C01820=1089.401,52.222,440.400,175.154,18.357,152.860
C01821=1089.407,52.472,440.384,175.156,18.358,152.860
C01822=1089.412,52.722,440.367,175.158,18.360,152.860
C01823=1089.418,52.971,440.351,175.160,18.362,152.860
C01824=1089.423,53.220,440.335,175.161,18.363,152.860
C01825=1089.429,53.469,440.319,175.163,18.365,152.860
C01826=1089.435,53.719,440.303,175.165,18.367,152.860
C01827=1089.441,53.969,440.287,175.167,18.368,152.860
C01828=1089.447,54.218,440.271,175.169,18.370,152.860
C01829=1089.453,54.467,440.255,175.171,18.372,152.860
C01830=1089.458,54.717,440.239,175.173,18.373,152.860
C01831=1089.464,54.966,440.223,175.175,18.375,152.860
C01832=1089.469,55.216,440.206,175.177,18.376,152.860
C01833=1089.475,55.465,440.190,175.178,18.378,152.860
C01834=1089.481,55.714,440.174,175.180,18.380,152.860
C01835=1089.486,55.964,440.158,175.182,18.381,152.860
C01836=1089.492,56.214,440.142,175.184,18.383,152.860
C01837=1089.498,56.463,440.126,175.186,18.385,152.860
C01838=1089.504,56.712,440.110,175.188,18.386,152.860
C01839=1089.510,56.961,440.094,175.189,18.388,152.860
C01840=1089.515,57.211,440.077,175.192,18.389,152.860
C01841=1089.521,57.460,440.061,175.193,18.391,152.860
C01842=1089.526,57.710,440.045,175.196,18.392,152.860
C01843=1089.532,57.959,440.029,175.197,18.394,152.860
C01844=1089.538,58.209,440.013,175.199,18.396,152.860
C01845=1089.544,58.458,439.996,175.201,18.397,152.860
C01846=1089.549,58.708,439.979,175.203,18.399,152.860
C01847=1089.555,58.957,439.963,175.205,18.400,152.859
C01848=1089.561,59.206,439.947,175.206,18.402,152.859
C01849=1089.567,59.456,439.931,175.209,18.403,152.859
C01850=1089.573,59.705,439.914,175.210,18.405,152.859
C01851=1089.579,59.954,439.898,175.213,18.407,152.859
C01852=1089.584,60.204,439.881,175.214,18.408,152.859
C01853=1089.590,60.453,439.865,175.217,18.410,152.859
C01854=1089.596,60.702,439.849,175.218,18.411,152.859
C01855=1089.602,60.951,439.833,175.221,18.413,152.859
C01856=1089.608,61.201,439.817,175.222,18.414,152.859
C01857=1089.613,61.450,439.800,175.224,18.415,152.859
C01858=1089.619,61.700,439.784,175.226,18.418,152.859
C01859=1089.625,61.949,439.767,175.228,18.419,152.859
C01860=1089.631,62.198,439.751,175.230,18.421,152.859
C01861=1089.636,62.448,439.734,175.232,18.422,152.859
C01862=1089.642,62.697,439.718,175.234,18.424,152.859
C01863=1089.648,62.947,439.702,175.235,18.425,152.859
C01864=1089.654,63.224,439.683,175.238,18.427,152.859
C01865=1089.661,63.501,439.665,175.240,18.429,152.859
C01866=1089.667,63.778,439.647,175.242,18.431,152.859
C01867=1089.674,64.055,439.629,175.244,18.432,152.859
C01868=1089.680,64.304,439.612,175.246,18.434,152.859
C01869=1089.685,64.554,439.596,175.248,18.435,152.859
C01870=1089.691,64.803,439.579,175.250,18.437,152.859
C01871=1089.697,65.052,439.562,175.252,18.438,152.858
C01872=1089.702,65.302,439.545,175.254,18.440,152.858
C01873=1089.708,65.551,439.529,175.256,18.441,152.858
C01874=1089.714,65.801,439.512,175.258,18.443,152.858
C01875=1089.720,66.050,439.496,175.260,18.444,152.858
C01876=1089.725,66.300,439.479,175.262,18.446,152.858
C01877=1089.731,66.548,439.462,175.264,18.447,152.858
C01878=1089.737,66.798,439.446,175.266,18.450,152.858
C01879=1089.742,67.047,439.429,175.268,18.451,152.858
C01880=1089.748,67.297,439.413,175.270,18.453,152.858
C01881=1089.753,67.546,439.396,175.271,18.454,152.858
C01882=1089.760,67.795,439.379,175.274,18.456,152.858
C01883=1089.765,68.045,439.362,175.275,18.457,152.858
C01884=1089.771,68.294,439.346,175.278,18.459,152.858
C01885=1089.776,68.544,439.329,175.279,18.460,152.858
C01886=1089.782,68.792,439.312,175.282,18.462,152.858
C01887=1089.788,69.043,439.295,175.283,18.463,152.858
C01888=1089.794,69.292,439.279,175.286,18.465,152.858
C01889=1089.799,69.542,439.262,175.287,18.466,152.858
C01890=1089.806,69.791,439.245,175.290,18.468,152.858
C01891=1089.811,70.040,439.228,175.291,18.469,152.858
C01892=1089.817,70.290,439.212,175.294,18.471,152.857
C01893=1089.822,70.539,439.194,175.295,18.473,152.858
C01894=1089.828,70.788,439.178,175.297,18.474,152.857
C01895=1089.833,71.038,439.161,175.299,18.476,152.857
C01896=1089.839,71.287,439.144,175.301,18.477,152.857
C01897=1089.845,71.536,439.127,175.303,18.478,152.857
C01898=1089.850,71.786,439.110,175.305,18.480,152.857
C01899=1089.856,72.034,439.093,175.307,18.482,152.857
C01900=1089.862,72.284,439.077,175.309,18.484,152.857
C01901=1089.867,72.534,439.060,175.311,18.485,152.857
C01902=1089.874,72.783,439.042,175.313,18.486,152.857
C01903=1089.879,73.033,439.026,175.315,18.488,152.857
C01904=1089.884,73.282,439.008,175.317,18.489,152.857
C01905=1089.890,73.531,438.992,175.319,18.491,152.857
C01906=1089.895,73.781,438.975,175.321,18.493,152.857
C01907=1089.902,74.030,438.958,175.323,18.494,152.857
C01908=1089.907,74.279,438.941,175.325,18.496,152.857
C01909=1089.912,74.528,438.923,175.327,18.497,152.857
C01910=1089.918,74.778,438.907,175.329,18.499,152.857
C01911=1089.924,75.027,438.890,175.331,18.500,152.857
C01912=1089.930,75.277,438.872,175.333,18.501,152.856
C01913=1089.936,75.526,438.855,175.335,18.503,152.856
C01914=1089.941,75.775,438.839,175.337,18.505,152.856
C01915=1089.947,76.024,438.821,175.339,18.506,152.856
C01916=1089.953,76.274,438.805,175.341,18.508,152.856
C01917=1089.958,76.523,438.787,175.343,18.509,152.856
C01918=1089.964,76.773,438.770,175.345,18.510,152.856
C01919=1089.970,77.022,438.752,175.347,18.512,152.856
C01920=1089.976,77.272,438.736,175.349,18.514,152.856
C01921=1089.981,77.521,438.719,175.352,18.515,152.856
C01922=1089.986,77.770,438.702,175.353,18.517,152.856
C01923=1089.992,78.019,438.685,175.355,18.518,152.856
C01924=1089.999,78.269,438.667,175.357,18.519,152.856
C01925=1090.004,78.518,438.650,175.360,18.521,152.855
C01926=1090.009,78.767,438.632,175.361,18.522,152.856
C01927=1090.015,79.017,438.616,175.364,18.524,152.855
C01928=1090.021,79.294,438.596,175.366,18.526,152.855
C01929=1090.028,79.571,438.577,175.367,18.527,152.855
C01930=1090.034,79.848,438.558,175.370,18.529,152.855
C01931=1090.040,80.124,438.539,175.372,18.531,152.855
C01932=1090.046,80.374,438.521,175.374,18.532,152.855
C01933=1090.051,80.623,438.504,175.376,18.533,152.855
C01934=1090.057,80.872,438.487,175.379,18.536,152.855
C01935=1090.062,81.121,438.469,175.380,18.537,152.855
C01936=1090.068,81.371,438.452,175.383,18.538,152.855
C01937=1090.073,81.620,438.435,175.384,18.539,152.855
C01938=1090.079,81.870,438.417,175.387,18.541,152.855
C01939=1090.084,82.119,438.400,175.388,18.542,152.855
C01940=1090.091,82.368,438.383,175.391,18.544,152.854
C01941=1090.096,82.617,438.366,175.392,18.546,152.855
C01942=1090.102,82.867,438.348,175.395,18.547,152.854
C01943=1090.108,83.117,438.331,175.396,18.548,152.854
C01944=1090.113,83.366,438.313,175.399,18.550,152.854
C01945=1090.119,83.615,438.296,175.401,18.552,152.854
C01946=1090.124,83.864,438.278,175.403,18.553,152.854
C01947=1090.130,84.114,438.261,175.405,18.554,152.854
C01948=1090.135,84.363,438.243,175.407,18.556,152.854
C01949=1090.141,84.612,438.226,175.410,18.557,152.854
C01950=1090.147,84.861,438.208,175.411,18.559,152.854
C01951=1090.153,85.111,438.190,175.413,18.560,152.854
C01952=1090.158,85.361,438.173,175.415,18.561,152.854
C01953=1090.163,85.610,438.156,175.418,18.563,152.853
C01954=1090.169,85.859,438.138,175.420,18.565,152.853
C01955=1090.175,86.108,438.120,175.421,18.566,152.853
C01956=1090.181,86.358,438.103,175.424,18.568,152.853
C01957=1090.186,86.607,438.085,175.426,18.569,152.853
C01958=1090.193,86.856,438.068,175.428,18.570,152.853
C01959=1090.198,87.106,438.051,175.430,18.571,152.853
C01960=1090.204,87.355,438.033,175.432,18.573,152.853
C01961=1090.210,87.604,438.016,175.434,18.574,152.853
C01962=1090.215,87.853,437.998,175.436,18.576,152.853
C01963=1090.221,88.102,437.980,175.439,18.578,152.853
C01964=1090.227,88.352,437.962,175.440,18.579,152.852
C01965=1090.232,88.601,437.945,175.443,18.580,152.852
C01966=1090.238,88.850,437.927,175.445,18.581,152.852
C01967=1090.244,89.100,437.909,175.447,18.583,152.852
C01968=1090.250,89.349,437.892,175.449,18.584,152.852
C01969=1090.255,89.598,437.874,175.451,18.586,152.852
C01970=1090.261,89.848,437.856,175.454,18.588,152.852
C01971=1090.266,90.097,437.838,175.455,18.589,152.852
C01972=1090.272,90.346,437.821,175.458,18.590,152.852
C01973=1090.278,90.596,437.803,175.459,18.591,152.852
C01974=1090.283,90.845,437.785,175.462,18.593,152.851
C01975=1090.289,91.095,437.767,175.464,18.594,152.851
C01976=1090.295,91.344,437.750,175.466,18.596,152.851
C01977=1090.300,91.593,437.732,175.469,18.597,152.851
C01978=1090.306,91.843,437.714,175.470,18.598,152.851
C01979=1090.311,92.092,437.696,175.473,18.600,152.851
C01980=1090.317,92.341,437.678,175.474,18.601,152.851
C01981=1090.323,92.591,437.660,175.477,18.603,152.851
C01982=1090.328,92.840,437.643,175.478,18.604,152.851
C01983=1090.334,93.088,437.625,175.481,18.606,152.851
C01984=1090.340,93.338,437.606,175.483,18.607,152.850
C01985=1090.345,93.587,437.588,175.485,18.608,152.850
C01986=1090.351,93.836,437.571,175.487,18.610,152.850
C01987=1090.357,94.086,437.553,175.489,18.611,152.850
C01988=1090.362,94.335,437.535,175.492,18.612,152.850
C01989=1090.368,94.585,437.517,175.494,18.614,152.850
C01990=1090.373,94.834,437.499,175.496,18.615,152.850
C01991=1090.379,95.083,437.481,175.498,18.617,152.850
C01992=1090.385,95.361,437.461,175.501,18.618,152.850
C01993=1090.391,95.637,437.440,175.503,18.620,152.849
C01994=1090.398,95.914,437.421,175.505,18.621,152.849
C01995=1090.404,96.190,437.401,175.507,18.623,152.849
C01996=1090.410,96.440,437.383,175.510,18.624,152.849
C01997=1090.415,96.690,437.365,175.512,18.625,152.849
C01998=1090.421,96.939,437.347,175.514,18.627,152.849
C01999=1090.427,97.188,437.328,175.517,18.628,152.849
C02000=1090.432,97.437,437.311,175.518,18.629,152.849
C02001=1090.438,97.687,437.292,175.521,18.631,152.848
C02002=1090.443,97.936,437.275,175.522,18.632,152.848
C02003=1090.450,98.185,437.256,175.525,18.634,152.848
C02004=1090.455,98.434,437.238,175.527,18.635,152.848
C02005=1090.461,98.684,437.220,175.529,18.636,152.848
C02006=1090.467,98.933,437.202,175.532,18.638,152.848
C02007=1090.472,99.183,437.183,175.533,18.639,152.848
C02008=1090.477,99.432,437.166,175.536,18.640,152.848
C02009=1090.484,99.681,437.147,175.538,18.642,152.848
C02010=1090.489,99.930,437.129,175.540,18.643,152.847
C02011=1090.495,100.180,437.111,175.542,18.645,152.847
C02012=1090.501,100.428,437.093,175.544,18.646,152.847
C02013=1090.507,100.678,437.075,175.547,18.647,152.847
C02014=1090.511,100.927,437.057,175.549,18.648,152.847
C02015=1090.518,101.176,437.038,175.551,18.649,152.847
C02016=1090.523,101.426,437.020,175.554,18.651,152.847
C02017=1090.529,101.675,437.001,175.556,18.653,152.847
C02018=1090.534,101.924,436.983,175.558,18.654,152.846
C02019=1090.540,102.174,436.965,175.560,18.655,152.846
C02020=1090.545,102.423,436.946,175.562,18.656,152.846
C02021=1090.551,102.672,436.928,175.564,18.658,152.846
C02022=1090.556,102.921,436.909,175.567,18.660,152.846
C02023=1090.562,103.171,436.891,175.569,18.661,152.846
C02024=1090.568,103.420,436.872,175.571,18.662,152.846
C02025=1090.574,103.669,436.855,175.574,18.664,152.846
C02026=1090.579,103.918,436.836,175.575,18.665,152.846
C02027=1090.585,104.168,436.818,175.578,18.666,152.845
C02028=1090.590,104.417,436.799,175.580,18.667,152.845
C02029=1090.596,104.666,436.781,175.582,18.669,152.845
C02030=1090.601,104.915,436.762,175.585,18.670,152.845
C02031=1090.607,105.165,436.744,175.586,18.671,152.845
C02032=1090.612,105.414,436.725,175.589,18.673,152.845
C02033=1090.618,105.663,436.707,175.591,18.674,152.845
C02034=1090.624,105.912,436.688,175.593,18.675,152.844
C02035=1090.630,106.161,436.670,175.596,18.676,152.844
C02036=1090.635,106.411,436.651,175.597,18.678,152.844
C02037=1090.640,106.660,436.632,175.600,18.679,152.844
C02038=1090.647,106.910,436.614,175.602,18.681,152.844
C02039=1090.652,107.158,436.596,175.604,18.682,152.844
C02040=1090.658,107.408,436.577,175.607,18.683,152.843
C02041=1090.663,107.657,436.559,175.609,18.684,152.843
C02042=1090.669,107.906,436.540,175.611,18.686,152.843
C02043=1090.675,108.156,436.522,175.614,18.687,152.843
C02044=1090.680,108.405,436.503,175.616,18.688,152.843
C02045=1090.686,108.654,436.484,175.618,18.689,152.843
C02046=1090.692,108.903,436.465,175.621,18.691,152.843
C02047=1090.697,109.152,436.447,175.622,18.692,152.843
C02048=1090.703,109.402,436.428,175.625,18.693,152.842
C02049=1090.708,109.651,436.409,175.627,18.695,152.842
C02050=1090.714,109.900,436.391,175.629,18.696,152.842
C02051=1090.720,110.150,436.372,175.632,18.697,152.842
C02052=1090.725,110.398,436.353,175.634,18.698,152.842
C02053=1090.731,110.648,436.334,175.636,18.699,152.842
C02054=1090.737,110.898,436.316,175.639,18.701,152.841
C02055=1090.743,111.146,436.298,175.641,18.702,152.841
C02056=1090.749,111.424,436.276,175.644,18.704,152.841
C02057=1090.755,111.700,436.256,175.645,18.705,152.841
C02058=1090.761,111.977,436.235,175.648,18.706,152.841
C02059=1090.768,112.255,436.214,175.651,18.707,152.841
C02060=1090.773,112.503,436.195,175.653,18.709,152.840
C02061=1090.779,112.753,436.176,175.656,18.711,152.840
C02062=1090.785,113.002,436.157,175.658,18.711,152.840
C02063=1090.790,113.251,436.138,175.660,18.713,152.840
C02064=1090.796,113.501,436.120,175.663,18.714,152.840
C02065=1090.801,113.750,436.101,175.665,18.715,152.840
C02066=1090.807,113.999,436.082,175.667,18.716,152.839
C02067=1090.813,114.248,436.063,175.670,18.718,152.839
C02068=1090.819,114.498,436.044,175.672,18.719,152.839
C02069=1090.824,114.746,436.025,175.674,18.720,152.839
C02070=1090.829,114.996,436.006,175.677,18.722,152.839
C02071=1090.835,115.245,435.986,175.678,18.723,152.839
C02072=1090.840,115.494,435.968,175.681,18.724,152.839
C02073=1090.846,115.744,435.949,175.683,18.725,152.838
C02074=1090.851,115.993,435.930,175.685,18.727,152.838
C02075=1090.856,116.242,435.911,175.688,18.728,152.838
C02076=1090.862,116.491,435.892,175.690,18.729,152.838
C02077=1090.868,116.741,435.873,175.692,18.730,152.838
C02078=1090.874,116.989,435.854,175.695,18.731,152.838
C02079=1090.879,117.239,435.835,175.697,18.733,152.837
C02080=1090.885,117.488,435.816,175.699,18.734,152.837
C02081=1090.890,117.737,435.797,175.701,18.736,152.837
C02082=1090.896,117.986,435.778,175.704,18.737,152.837
C02083=1090.901,118.236,435.758,175.706,18.738,152.837
C02084=1090.907,118.485,435.739,175.709,18.739,152.837
C02085=1090.912,118.734,435.720,175.711,18.740,152.836
C02086=1090.918,118.983,435.701,175.714,18.742,152.836
C02087=1090.924,119.233,435.682,175.716,18.743,152.836
C02088=1090.929,119.481,435.662,175.718,18.744,152.836
C02089=1090.935,119.730,435.643,175.721,18.746,152.836
C02090=1090.940,119.980,435.624,175.723,18.746,152.836
C02091=1090.946,120.229,435.604,175.725,18.748,152.835
C02092=1090.951,120.478,435.585,175.728,18.749,152.835
C02093=1090.957,120.727,435.566,175.729,18.750,152.835
C02094=1090.962,120.977,435.547,175.732,18.751,152.835
C02095=1090.968,121.226,435.528,175.735,18.753,152.835
C02096=1090.974,121.476,435.509,175.736,18.754,152.835
C02097=1090.979,121.724,435.489,175.739,18.755,152.834
C02098=1090.985,121.973,435.470,175.742,18.756,152.834
C02099=1090.991,122.223,435.450,175.744,18.757,152.834
C02100=1090.996,122.472,435.431,175.746,18.759,152.834
C02101=1091.002,122.722,435.412,175.749,18.760,152.834
C02102=1091.007,122.970,435.392,175.751,18.761,152.833
C02103=1091.013,123.219,435.373,175.753,18.762,152.833
C02104=1091.019,123.469,435.354,175.756,18.763,152.833
C02105=1091.024,123.718,435.335,175.758,18.765,152.833
C02106=1091.029,123.968,435.315,175.760,18.766,152.833
C02107=1091.035,124.216,435.295,175.763,18.767,152.833
C02108=1091.040,124.465,435.276,175.765,18.768,152.832
C02109=1091.046,124.715,435.257,175.767,18.769,152.832
C02110=1091.052,124.963,435.237,175.770,18.770,152.832
C02111=1091.058,125.213,435.218,175.773,18.772,152.832
C02112=1091.064,125.462,435.198,175.775,18.773,152.831
C02113=1091.069,125.712,435.179,175.777,18.774,152.831
C02114=1091.075,125.961,435.159,175.780,18.775,152.831
C02115=1091.080,126.209,435.140,175.782,18.776,152.831
C02116=1091.086,126.459,435.121,175.784,18.777,152.831
C02117=1091.092,126.708,435.101,175.787,18.778,152.831
C02118=1091.097,126.957,435.081,175.789,18.780,152.830
C02119=1091.103,127.206,435.061,175.792,18.781,152.830
C02120=1091.110,127.483,435.040,175.795,18.782,152.830
C02121=1091.116,127.760,435.018,175.797,18.783,152.830
C02122=1091.122,128.037,434.996,175.800,18.784,152.829
C02123=1091.128,128.315,434.975,175.803,18.786,152.829
C02124=1091.134,128.563,434.955,175.805,18.787,152.829
C02125=1091.139,128.812,434.936,175.807,18.788,152.829
C02126=1091.145,129.061,434.916,175.810,18.789,152.829
C02127=1091.151,129.311,434.897,175.813,18.790,152.828
C02128=1091.157,129.559,434.877,175.815,18.791,152.828
C02129=1091.163,129.809,434.857,175.817,18.792,152.828
C02130=1091.168,130.058,434.837,175.820,18.794,152.828
C02131=1091.174,130.307,434.818,175.822,18.794,152.828
C02132=1091.179,130.556,434.798,175.825,18.795,152.827
C02133=1091.185,130.806,434.778,175.827,18.796,152.827
C02134=1091.191,131.055,434.758,175.830,18.798,152.827
C02135=1091.197,131.304,434.739,175.832,18.799,152.827
C02136=1091.202,131.553,434.719,175.834,18.800,152.826
C02137=1091.208,131.803,434.699,175.837,18.801,152.826
C02138=1091.214,132.051,434.679,175.840,18.802,152.826
C02139=1091.219,132.301,434.660,175.842,18.803,152.826
C02140=1091.225,132.550,434.640,175.844,18.804,152.826
C02141=1091.231,132.799,434.620,175.847,18.806,152.825
C02142=1091.236,133.048,434.600,175.850,18.807,152.825
C02143=1091.242,133.297,434.580,175.852,18.807,152.825
C02144=1091.247,133.547,434.561,175.854,18.809,152.825
C02145=1091.253,133.795,434.541,175.857,18.810,152.825
C02146=1091.259,134.045,434.520,175.859,18.811,152.824
C02147=1091.264,134.294,434.501,175.861,18.812,152.824
C02148=1091.270,134.543,434.480,175.864,18.813,152.824
C02149=1091.276,134.792,434.460,175.867,18.814,152.824
C02150=1091.281,135.041,434.441,175.869,18.815,152.823
C02151=1091.286,135.291,434.420,175.871,18.816,152.823
C02152=1091.292,135.539,434.401,175.874,18.818,152.823
C02153=1091.297,135.789,434.381,175.877,18.819,152.823
C02154=1091.303,136.038,434.361,175.879,18.819,152.823
C02155=1091.309,136.287,434.341,175.881,18.821,152.822
C02156=1091.315,136.536,434.320,175.884,18.822,152.822
C02157=1091.320,136.785,434.301,175.887,18.823,152.822
C02158=1091.326,137.034,434.280,175.889,18.824,152.822
C02159=1091.332,137.283,434.260,175.891,18.825,152.821
C02160=1091.337,137.532,434.240,175.894,18.826,152.821
C02161=1091.343,137.782,434.221,175.897,18.827,152.821
C02162=1091.348,138.031,434.200,175.899,18.829,152.821
C02163=1091.354,138.280,434.180,175.901,18.829,152.820
C02164=1091.360,138.529,434.160,175.904,18.830,152.820
C02165=1091.365,138.778,434.140,175.907,18.832,152.820
C02166=1091.371,139.027,434.120,175.909,18.833,152.820
C02167=1091.377,139.277,434.099,175.911,18.833,152.820
C02168=1091.382,139.526,434.079,175.914,18.835,152.819
C02169=1091.388,139.775,434.059,175.917,18.836,152.819
C02170=1091.393,140.024,434.038,175.919,18.837,152.819
C02171=1091.399,140.273,434.018,175.921,18.837,152.819
C02172=1091.404,140.522,433.998,175.924,18.839,152.818
C02173=1091.410,140.771,433.978,175.927,18.840,152.818
C02174=1091.415,141.020,433.958,175.929,18.841,152.818
C02175=1091.421,141.269,433.938,175.932,18.842,152.818
C02176=1091.427,141.518,433.918,175.934,18.843,152.817
C02177=1091.432,141.768,433.897,175.937,18.844,152.817
C02178=1091.438,142.016,433.877,175.939,18.845,152.817
C02179=1091.444,142.266,433.856,175.942,18.847,152.817
C02180=1091.449,142.515,433.836,175.944,18.847,152.817
C02181=1091.455,142.764,433.816,175.947,18.848,152.816
C02182=1091.460,143.013,433.795,175.950,18.849,152.816
C02183=1091.465,143.262,433.775,175.952,18.850,152.816
C02184=1091.472,143.539,433.752,175.955,18.852,152.815
C02185=1091.478,143.816,433.730,175.958,18.853,152.815
C02186=1091.485,144.093,433.707,175.961,18.854,152.815
C02187=1091.490,144.369,433.684,175.963,18.855,152.815
C02188=1091.497,144.619,433.664,175.966,18.856,152.814
C02189=1091.502,144.868,433.643,175.969,18.857,152.814
C02190=1091.507,145.117,433.622,175.972,18.858,152.814
C02191=1091.513,145.366,433.602,175.973,18.859,152.814
C02192=1091.519,145.615,433.582,175.976,18.860,152.813
C02193=1091.524,145.864,433.561,175.979,18.861,152.813
C02194=1091.530,146.114,433.540,175.982,18.862,152.813
C02195=1091.536,146.363,433.520,175.984,18.863,152.813
C02196=1091.541,146.611,433.499,175.986,18.864,152.812
C02197=1091.547,146.860,433.479,175.989,18.865,152.812
C02198=1091.553,147.109,433.459,175.992,18.866,152.812
C02199=1091.558,147.359,433.438,175.995,18.867,152.812
C02200=1091.564,147.608,433.417,175.997,18.868,152.811
C02201=1091.569,147.857,433.397,175.999,18.869,152.811
C02202=1091.575,148.105,433.376,176.002,18.870,152.811
C02203=1091.581,148.355,433.355,176.005,18.871,152.811
C02204=1091.586,148.604,433.335,176.008,18.872,152.810
C02205=1091.592,148.853,433.314,176.010,18.873,152.810
C02206=1091.597,149.103,433.293,176.013,18.874,152.810
C02207=1091.603,149.351,433.273,176.015,18.875,152.810
C02208=1091.609,149.601,433.252,176.018,18.876,152.809
C02209=1091.614,149.850,433.231,176.021,18.877,152.809
C02210=1091.620,150.098,433.210,176.023,18.878,152.809
C02211=1091.625,150.347,433.189,176.026,18.879,152.808
C02212=1091.631,150.597,433.169,176.028,18.880,152.808
C02213=1091.636,150.846,433.148,176.031,18.881,152.808
C02214=1091.642,151.095,433.127,176.033,18.882,152.808
C02215=1091.648,151.344,433.107,176.036,18.883,152.807
C02216=1091.654,151.593,433.086,176.039,18.884,152.807
C02217=1091.659,151.842,433.065,176.042,18.885,152.807
C02218=1091.664,152.091,433.044,176.044,18.886,152.807
C02219=1091.670,152.340,433.023,176.046,18.887,152.806
C02220=1091.676,152.589,433.002,176.049,18.888,152.806
C02221=1091.681,152.839,432.981,176.052,18.889,152.806
C02222=1091.687,153.087,432.960,176.055,18.890,152.806
C02223=1091.692,153.336,432.939,176.057,18.891,152.805
C02224=1091.698,153.586,432.919,176.060,18.891,152.805
C02225=1091.703,153.834,432.897,176.062,18.893,152.805
C02226=1091.709,154.084,432.877,176.065,18.894,152.804
C02227=1091.715,154.333,432.855,176.068,18.895,152.804
C02228=1091.720,154.582,432.835,176.071,18.896,152.804
C02229=1091.726,154.830,432.813,176.073,18.897,152.804
C02230=1091.731,155.080,432.792,176.075,18.898,152.803
C02231=1091.737,155.329,432.771,176.078,18.898,152.803
C02232=1091.742,155.578,432.750,176.081,18.899,152.803
C02233=1091.748,155.827,432.729,176.084,18.900,152.803
C02234=1091.754,156.076,432.708,176.087,18.902,152.802
C02235=1091.759,156.325,432.687,176.089,18.903,152.802
C02236=1091.765,156.575,432.666,176.092,18.904,152.802
C02237=1091.771,156.823,432.645,176.094,18.904,152.802
C02238=1091.776,157.072,432.624,176.097,18.905,152.801
C02239=1091.782,157.321,432.603,176.100,18.906,152.801
C02240=1091.787,157.571,432.582,176.102,18.907,152.801
C02241=1091.793,157.819,432.561,176.105,18.908,152.800
C02242=1091.799,158.068,432.539,176.108,18.909,152.800
C02243=1091.804,158.317,432.519,176.111,18.910,152.800
C02244=1091.809,158.566,432.497,176.113,18.911,152.799
C02245=1091.815,158.816,432.476,176.116,18.912,152.799
C02246=1091.821,159.065,432.455,176.118,18.913,152.799
C02247=1091.827,159.314,432.433,176.121,18.914,152.799
C02248=1091.833,159.590,432.409,176.124,18.915,152.798
C02249=1091.839,159.867,432.387,176.127,18.916,152.798
C02250=1091.845,160.143,432.363,176.131,18.917,152.798
C02251=1091.852,160.420,432.339,176.134,18.918,152.797
C02252=1091.857,160.669,432.318,176.136,18.919,152.797
C02253=1091.863,160.918,432.296,176.138,18.920,152.797
C02254=1091.869,161.167,432.275,176.141,18.920,152.796
C02255=1091.874,161.416,432.253,176.144,18.921,152.796
C02256=1091.879,161.666,432.232,176.147,18.922,152.796
C02257=1091.885,161.914,432.211,176.149,18.924,152.796
C02258=1091.890,162.164,432.189,176.152,18.925,152.795
C02259=1091.896,162.412,432.168,176.155,18.925,152.795
C02260=1091.901,162.661,432.147,176.158,18.926,152.795
C02261=1091.907,162.911,432.125,176.161,18.927,152.794
C02262=1091.912,163.159,432.104,176.163,18.928,152.794
C02263=1091.918,163.408,432.082,176.165,18.929,152.794
C02264=1091.923,163.657,432.060,176.168,18.930,152.794
C02265=1091.928,163.906,432.039,176.171,18.931,152.793
C02266=1091.934,164.156,432.017,176.174,18.932,152.793
C02267=1091.939,164.404,431.996,176.177,18.933,152.793
C02268=1091.944,164.653,431.974,176.179,18.934,152.792
C02269=1091.950,164.902,431.952,176.182,18.935,152.792
C02270=1091.956,165.151,431.931,176.185,18.936,152.792
C02271=1091.961,165.400,431.909,176.187,18.937,152.792
C02272=1091.967,165.649,431.888,176.190,18.938,152.791
C02273=1091.972,165.898,431.865,176.193,18.939,152.791
C02274=1091.978,166.148,431.845,176.196,18.939,152.791
C02275=1091.982,166.396,431.823,176.198,18.940,152.790
C02276=1091.989,166.646,431.801,176.201,18.942,152.790
C02277=1091.993,166.894,431.780,176.204,18.943,152.790
C02278=1092.000,167.144,431.758,176.207,18.943,152.789
C02279=1092.005,167.392,431.737,176.210,18.944,152.789
C02280=1092.011,167.642,431.714,176.212,18.946,152.789
C02281=1092.016,167.890,431.693,176.215,18.946,152.789
C02282=1092.022,168.140,431.671,176.217,18.947,152.788
C02283=1092.027,168.388,431.650,176.220,18.948,152.788
C02284=1092.033,168.638,431.627,176.223,18.949,152.788
C02285=1092.038,168.886,431.606,176.226,18.950,152.787
C02286=1092.044,169.136,431.584,176.229,18.951,152.787
C02287=1092.049,169.384,431.563,176.232,18.951,152.787
C02288=1092.055,169.633,431.540,176.234,18.952,152.786
C02289=1092.060,169.882,431.518,176.237,18.954,152.786
C02290=1092.066,170.131,431.496,176.240,18.954,152.786
C02291=1092.071,170.380,431.475,176.243,18.955,152.786
C02292=1092.077,170.629,431.453,176.246,18.956,152.785
C02293=1092.083,170.878,431.431,176.249,18.957,152.785
C02294=1092.088,171.127,431.409,176.251,18.958,152.785
C02295=1092.093,171.377,431.387,176.253,18.958,152.784
C02296=1092.099,171.625,431.365,176.256,18.959,152.784
C02297=1092.105,171.874,431.343,176.259,18.961,152.784
C02298=1092.110,172.123,431.321,176.262,18.961,152.783
C02299=1092.116,172.372,431.299,176.265,18.962,152.783
C02300=1092.122,172.621,431.278,176.268,18.963,152.783
C02301=1092.127,172.869,431.255,176.271,18.964,152.782
C02302=1092.133,173.119,431.233,176.274,18.965,152.782
C02303=1092.138,173.368,431.211,176.276,18.966,152.782
C02304=1092.143,173.617,431.189,176.279,18.967,152.782
C02305=1092.150,173.866,431.167,176.282,18.968,152.781
C02306=1092.155,174.114,431.145,176.285,18.969,152.781
C02307=1092.161,174.364,431.123,176.288,18.969,152.780
C02308=1092.166,174.613,431.101,176.291,18.970,152.780
C02309=1092.171,174.861,431.079,176.294,18.971,152.780
C02310=1092.177,175.111,431.057,176.296,18.972,152.780
C02311=1092.183,175.360,431.035,176.298,18.972,152.779
C02312=1092.189,175.636,431.011,176.302,18.973,152.779
C02313=1092.195,175.911,430.986,176.305,18.974,152.778
C02314=1092.202,176.188,430.961,176.308,18.975,152.778
C02315=1092.208,176.464,430.936,176.312,18.976,152.778
C02316=1092.214,176.714,430.915,176.315,18.977,152.777
C02317=1092.219,176.963,430.892,176.317,18.978,152.777
C02318=1092.224,177.211,430.870,176.320,18.979,152.777
C02319=1092.231,177.460,430.848,176.323,18.979,152.776
C02320=1092.236,177.710,430.825,176.326,18.980,152.776
C02321=1092.241,177.958,430.803,176.328,18.981,152.776
C02322=1092.247,178.207,430.781,176.331,18.982,152.775
C02323=1092.253,178.456,430.759,176.334,18.983,152.775
C02324=1092.259,178.705,430.736,176.337,18.983,152.775
C02325=1092.264,178.954,430.715,176.340,18.984,152.774
C02326=1092.270,179.203,430.692,176.343,18.985,152.774
C02327=1092.275,179.452,430.669,176.346,18.986,152.774
C02328=1092.282,179.701,430.647,176.349,18.987,152.773
C02329=1092.287,179.950,430.625,176.352,18.988,152.773
C02330=1092.292,180.199,430.602,176.355,18.988,152.773
C02331=1092.298,180.448,430.581,176.357,18.989,152.772
C02332=1092.304,180.697,430.558,176.360,18.990,152.772
C02333=1092.310,180.946,430.535,176.363,18.991,152.771
C02334=1092.316,181.194,430.514,176.366,18.992,152.771
C02335=1092.321,181.443,430.491,176.369,18.992,152.771
C02336=1092.327,181.692,430.468,176.372,18.993,152.770
C02337=1092.332,181.941,430.445,176.375,18.994,152.770
C02338=1092.339,182.190,430.423,176.378,18.995,152.770
C02339=1092.344,182.439,430.401,176.381,18.995,152.769
C02340=1092.349,182.688,430.378,176.384,18.996,152.769
C02341=1092.355,182.937,430.355,176.387,18.997,152.769
C02342=1092.361,183.186,430.334,176.390,18.998,152.768
C02343=1092.367,183.435,430.311,176.393,18.998,152.768
C02344=1092.373,183.684,430.288,176.395,19.000,152.768
C02345=1092.378,183.933,430.266,176.398,19.000,152.767
C02346=1092.384,184.181,430.244,176.401,19.001,152.767
C02347=1092.390,184.430,430.221,176.404,19.001,152.766
C02348=1092.396,184.679,430.198,176.407,19.003,152.766
C02349=1092.401,184.928,430.175,176.410,19.003,152.766
C02350=1092.407,185.177,430.152,176.413,19.004,152.765
C02351=1092.412,185.426,430.130,176.416,19.004,152.765
C02352=1092.418,185.675,430.107,176.419,19.006,152.765
C02353=1092.423,185.924,430.085,176.422,19.006,152.764
C02354=1092.429,186.173,430.062,176.425,19.007,152.764
C02355=1092.434,186.422,430.039,176.428,19.008,152.764
C02356=1092.440,186.670,430.016,176.430,19.009,152.763
C02357=1092.445,186.919,429.993,176.433,19.010,152.763
C02358=1092.451,187.168,429.971,176.436,19.010,152.763
C02359=1092.456,187.417,429.948,176.439,19.012,152.762
C02360=1092.461,187.666,429.925,176.442,19.012,152.762
C02361=1092.467,187.915,429.902,176.445,19.013,152.762
C02362=1092.473,188.164,429.879,176.448,19.014,152.761
C02363=1092.478,188.412,429.856,176.451,19.015,152.761
C02364=1092.484,188.661,429.833,176.454,19.016,152.761
C02365=1092.489,188.910,429.810,176.457,19.016,152.760
C02366=1092.495,189.160,429.788,176.460,19.017,152.760
C02367=1092.500,189.409,429.764,176.462,19.018,152.760
C02368=1092.506,189.658,429.742,176.465,19.019,152.759
C02369=1092.511,189.906,429.719,176.468,19.020,152.759
C02370=1092.517,190.155,429.696,176.471,19.021,152.759
C02371=1092.522,190.404,429.673,176.474,19.021,152.758
C02372=1092.528,190.653,429.650,176.477,19.022,152.758
C02373=1092.533,190.902,429.627,176.480,19.023,152.757
C02374=1092.539,191.151,429.604,176.483,19.024,152.757
C02375=1092.544,191.400,429.581,176.486,19.024,152.757
C02376=1092.550,191.675,429.555,176.490,19.025,152.756
C02377=1092.557,191.951,429.530,176.492,19.027,152.756
C02378=1092.563,192.227,429.504,176.496,19.028,152.756
C02379=1092.569,192.503,429.478,176.499,19.028,152.755
C02380=1092.575,192.751,429.455,176.502,19.029,152.755
C02381=1092.580,193.000,429.432,176.505,19.030,152.754
C02382=1092.585,193.249,429.409,176.508,19.031,152.754
C02383=1092.591,193.498,429.386,176.511,19.031,152.754
C02384=1092.597,193.747,429.363,176.514,19.032,152.753
C02385=1092.603,193.996,429.340,176.517,19.033,152.753
C02386=1092.608,194.245,429.316,176.520,19.033,152.753
C02387=1092.614,194.493,429.293,176.523,19.034,152.752
C02388=1092.619,194.742,429.270,176.526,19.035,152.752
C02389=1092.625,194.991,429.247,176.530,19.036,152.751
C02390=1092.630,195.240,429.223,176.533,19.037,152.751
C02391=1092.636,195.489,429.200,176.535,19.038,152.751
C02392=1092.642,195.737,429.177,176.538,19.039,152.750
C02393=1092.648,195.986,429.154,176.541,19.039,152.750
C02394=1092.653,196.236,429.130,176.544,19.040,152.750
C02395=1092.658,196.484,429.107,176.547,19.041,152.749
C02396=1092.664,196.733,429.084,176.550,19.041,152.749
C02397=1092.669,196.982,429.060,176.553,19.042,152.749
C02398=1092.675,197.231,429.037,176.556,19.043,152.748
C02399=1092.681,197.480,429.014,176.559,19.044,152.748
C02400=1092.687,197.729,428.990,176.562,19.044,152.747
C02401=1092.692,197.978,428.967,176.565,19.045,152.747
C02402=1092.698,198.227,428.944,176.569,19.046,152.747
C02403=1092.704,198.475,428.920,176.572,19.047,152.746
C02404=1092.709,198.724,428.896,176.575,19.048,152.746
C02405=1092.715,198.973,428.873,176.578,19.049,152.746
C02406=1092.721,199.222,428.850,176.581,19.049,152.745
C02407=1092.726,199.471,428.826,176.584,19.050,152.745
C02408=1092.732,199.719,428.803,176.587,19.051,152.744
C02409=1092.738,199.968,428.780,176.590,19.051,152.744
C02410=1092.743,200.217,428.756,176.593,19.052,152.744
C02411=1092.749,200.466,428.732,176.596,19.053,152.743
C02412=1092.754,200.715,428.709,176.599,19.053,152.743
C02413=1092.760,200.964,428.685,176.602,19.054,152.742
C02414=1092.766,201.212,428.662,176.605,19.055,152.742
C02415=1092.771,201.461,428.638,176.608,19.056,152.742
C02416=1092.777,201.710,428.615,176.611,19.057,152.741
C02417=1092.784,201.959,428.591,176.614,19.058,152.741
C02418=1092.789,202.208,428.567,176.617,19.058,152.741
C02419=1092.795,202.456,428.544,176.620,19.059,152.740
C02420=1092.800,202.706,428.520,176.623,19.059,152.740
C02421=1092.806,202.954,428.496,176.626,19.060,152.739
C02422=1092.811,203.203,428.473,176.629,19.061,152.739
C02423=1092.817,203.451,428.449,176.633,19.062,152.739
C02424=1092.823,203.701,428.425,176.636,19.063,152.738
C02425=1092.828,203.950,428.401,176.639,19.063,152.738
C02426=1092.834,204.198,428.377,176.642,19.064,152.737
C02427=1092.839,204.447,428.354,176.645,19.065,152.737
C02428=1092.845,204.696,428.330,176.648,19.066,152.737
C02429=1092.850,204.944,428.306,176.651,19.066,152.736
C02430=1092.855,205.193,428.282,176.654,19.067,152.736
C02431=1092.862,205.442,428.258,176.657,19.068,152.735
C02432=1092.867,205.691,428.234,176.660,19.069,152.735
C02433=1092.873,205.940,428.211,176.663,19.070,152.735
C02434=1092.878,206.188,428.187,176.666,19.071,152.734
C02435=1092.883,206.437,428.163,176.669,19.071,152.734
C02436=1092.890,206.686,428.139,176.672,19.072,152.734
C02437=1092.895,206.935,428.115,176.675,19.073,152.733
C02438=1092.900,207.184,428.091,176.679,19.074,152.733
C02439=1092.906,207.432,428.067,176.682,19.075,152.732
C02440=1092.929,208.451,427.969,176.741,19.102,152.728
C02441=1092.937,208.827,427.932,176.746,19.104,152.727
C02442=1092.946,209.204,427.896,176.750,19.107,152.727
C02443=1092.955,209.581,427.858,176.755,19.109,152.727
C02444=1092.963,209.957,427.822,176.759,19.112,152.727
C02445=1092.969,210.206,427.797,176.762,19.113,152.727
C02446=1092.974,210.455,427.773,176.765,19.115,152.726
C02447=1092.980,210.703,427.748,176.768,19.117,152.726
C02448=1092.986,210.952,427.724,176.771,19.119,152.726
C02449=1092.991,211.201,427.700,176.774,19.120,152.726
C02450=1092.997,211.450,427.675,176.777,19.121,152.726
C02451=1093.002,211.699,427.651,176.780,19.124,152.726
C02452=1093.008,211.947,427.626,176.782,19.125,152.726
C02453=1093.014,212.196,427.601,176.786,19.127,152.725
C02454=1093.019,212.445,427.577,176.789,19.128,152.725
C02455=1093.024,212.693,427.553,176.792,19.130,152.725
C02456=1093.030,212.943,427.528,176.795,19.132,152.725
C02457=1093.036,213.191,427.503,176.798,19.134,152.725
C02458=1093.042,213.440,427.478,176.801,19.135,152.724
C02459=1093.047,213.688,427.454,176.803,19.137,152.724
C02460=1093.053,213.938,427.430,176.807,19.139,152.724
C02461=1093.058,214.186,427.405,176.809,19.140,152.724
C02462=1093.064,214.434,427.380,176.813,19.142,152.724
C02463=1093.070,214.684,427.356,176.815,19.144,152.724
C02464=1093.075,214.932,427.331,176.819,19.145,152.723
C02465=1093.081,215.181,427.306,176.821,19.147,152.723
C02466=1093.086,215.429,427.282,176.824,19.149,152.723
C02467=1093.091,215.678,427.257,176.827,19.150,152.723
C02468=1093.097,215.927,427.232,176.831,19.152,152.723
C02469=1093.103,216.176,427.207,176.833,19.154,152.723
C02470=1093.108,216.425,427.183,176.837,19.156,152.722
C02471=1093.114,216.673,427.158,176.839,19.157,152.722
C02472=1093.120,216.922,427.133,176.842,19.159,152.722
C02473=1093.126,217.170,427.108,176.845,19.161,152.722
C02474=1093.131,217.420,427.083,176.848,19.162,152.722
C02475=1093.136,217.668,427.058,176.851,19.164,152.722
C02476=1093.142,217.917,427.033,176.854,19.165,152.722
C02477=1093.148,218.166,427.009,176.857,19.168,152.721
C02478=1093.154,218.414,426.984,176.860,19.169,152.721
C02479=1093.159,218.663,426.960,176.863,19.171,152.721
C02480=1093.164,218.912,426.934,176.866,19.173,152.721
C02481=1093.170,219.160,426.909,176.869,19.175,152.721
C02482=1093.176,219.409,426.884,176.872,19.176,152.721
C02483=1093.181,219.658,426.860,176.875,19.178,152.720
C02484=1093.187,219.906,426.834,176.878,19.179,152.720
C02485=1093.193,220.155,426.808,176.881,19.181,152.720
C02486=1093.198,220.404,426.784,176.884,19.183,152.720
C02487=1093.204,220.653,426.759,176.887,19.185,152.720
C02488=1093.210,220.901,426.735,176.890,19.186,152.720
C02489=1093.215,221.150,426.709,176.893,19.188,152.720
C02490=1093.221,221.398,426.684,176.896,19.189,152.719
C02491=1093.227,221.647,426.659,176.899,19.192,152.719
C02492=1093.233,221.896,426.634,176.902,19.193,152.719
C02493=1093.241,222.277,426.595,176.907,19.196,152.719
C02494=1093.250,222.657,426.556,176.911,19.198,152.718
C02495=1093.258,223.038,426.518,176.916,19.201,152.718
C02496=1093.267,223.418,426.480,176.921,19.204,152.718
C02497=1093.272,223.667,426.454,176.923,19.205,152.718
C02498=1093.278,223.915,426.429,176.927,19.207,152.718
C02499=1093.283,224.164,426.403,176.929,19.209,152.718
C02500=1093.289,224.412,426.378,176.933,19.211,152.717
C02501=1093.294,224.662,426.353,176.935,19.212,152.717
C02502=1093.300,224.910,426.328,176.939,19.214,152.717
C02503=1093.305,225.159,426.302,176.941,19.216,152.717
C02504=1093.311,225.407,426.277,176.945,19.218,152.717
C02505=1093.317,225.656,426.252,176.947,19.219,152.717
C02506=1093.322,225.904,426.226,176.950,19.221,152.717
C02507=1093.328,226.154,426.201,176.953,19.223,152.716
C02508=1093.334,226.403,426.176,176.957,19.225,152.716
C02509=1093.339,226.651,426.151,176.960,19.227,152.716
C02510=1093.345,226.900,426.125,176.963,19.228,152.716
C02511=1093.351,227.148,426.099,176.966,19.230,152.716
C02512=1093.356,227.397,426.074,176.968,19.232,152.716
C02513=1093.362,227.645,426.048,176.972,19.233,152.715
C02514=1093.368,227.894,426.022,176.975,19.235,152.715
C02515=1093.373,228.142,425.997,176.978,19.237,152.715
C02516=1093.379,228.391,425.972,176.981,19.238,152.715
C02517=1093.385,228.640,425.946,176.984,19.240,152.715
C02518=1093.390,228.889,425.920,176.986,19.242,152.715
C02519=1093.395,229.137,425.895,176.990,19.244,152.715
C02520=1093.401,229.386,425.869,176.993,19.245,152.714
C02521=1093.407,229.635,425.843,176.996,19.247,152.714
C02522=1093.413,229.883,425.818,176.999,19.249,152.714
C02523=1093.418,230.132,425.793,177.002,19.251,152.714
C02524=1093.424,230.380,425.767,177.005,19.253,152.714
C02525=1093.430,230.629,425.741,177.008,19.254,152.714
C02526=1093.435,230.878,425.715,177.011,19.256,152.713
C02527=1093.441,231.126,425.690,177.014,19.258,152.713
C02528=1093.446,231.375,425.664,177.017,19.260,152.713
C02529=1093.452,231.624,425.638,177.020,19.261,152.713
C02530=1093.458,231.872,425.612,177.023,19.263,152.713
C02531=1093.463,232.121,425.587,177.027,19.265,152.713
C02532=1093.468,232.370,425.561,177.029,19.267,152.713
C02533=1093.474,232.619,425.535,177.033,19.269,152.712
C02534=1093.480,232.867,425.510,177.035,19.270,152.712
C02535=1093.486,233.116,425.483,177.038,19.272,152.712
C02536=1093.491,233.364,425.457,177.042,19.275,152.712
C02537=1093.497,233.612,425.432,177.045,19.276,152.712
C02538=1093.502,233.861,425.406,177.048,19.278,152.712
C02539=1093.508,234.110,425.380,177.050,19.280,152.712
C02540=1093.514,234.359,425.354,177.054,19.282,152.712
C02541=1093.519,234.607,425.328,177.056,19.283,152.711
C02542=1093.525,234.855,425.302,177.060,19.285,152.711
C02543=1093.531,235.104,425.276,177.063,19.287,152.711
C02544=1093.536,235.353,425.250,177.066,19.289,152.711
C02545=1093.544,235.725,425.211,177.071,19.291,152.711
C02546=1093.553,236.097,425.172,177.075,19.294,152.711
C02547=1093.561,236.469,425.134,177.079,19.297,152.710
C02548=1093.569,236.840,425.094,177.084,19.300,152.710
C02549=1093.575,237.089,425.068,177.087,19.301,152.710
C02550=1093.580,237.338,425.042,177.090,19.303,152.710
C02551=1093.586,237.587,425.015,177.094,19.305,152.710
C02552=1093.592,237.835,424.990,177.096,19.307,152.710
C02553=1093.597,238.083,424.963,177.100,19.309,152.709
C02554=1093.603,238.332,424.938,177.102,19.310,152.709
C02555=1093.609,238.580,424.911,177.106,19.313,152.709
C02556=1093.614,238.829,424.885,177.109,19.315,152.709
C02557=1093.620,239.078,424.858,177.112,19.316,152.709
C02558=1093.625,239.327,424.832,177.115,19.318,152.709
C02559=1093.631,239.575,424.806,177.117,19.320,152.709
C02560=1093.637,239.823,424.779,177.121,19.322,152.709
C02561=1093.642,240.072,424.753,177.124,19.323,152.708
C02562=1093.648,240.321,424.727,177.127,19.325,152.708
C02563=1093.654,240.570,424.701,177.130,19.327,152.708
C02564=1093.659,240.818,424.674,177.134,19.329,152.708
C02565=1093.665,241.066,424.647,177.136,19.331,152.708
C02566=1093.671,241.315,424.621,177.140,19.333,152.708
C02567=1093.676,241.564,424.595,177.142,19.334,152.708
C02568=1093.681,241.812,424.569,177.145,19.336,152.707
C02569=1093.688,242.061,424.542,177.149,19.339,152.707
C02570=1093.693,242.310,424.515,177.152,19.340,152.707
C02571=1093.699,242.558,424.489,177.155,19.342,152.707
C02572=1093.705,242.807,424.463,177.158,19.344,152.707
C02573=1093.711,243.055,424.436,177.161,19.346,152.707
C02574=1093.716,243.304,424.410,177.164,19.347,152.707
C02575=1093.722,243.552,424.383,177.167,19.349,152.706
C02576=1093.727,243.800,424.357,177.170,19.351,152.706
C02577=1093.732,244.049,424.330,177.173,19.353,152.706
C02578=1093.738,244.297,424.303,177.176,19.355,152.706
C02579=1093.744,244.546,424.277,177.179,19.357,152.706
C02580=1093.749,244.795,424.251,177.183,19.359,152.706
C02581=1093.755,245.043,424.224,177.185,19.361,152.706
C02582=1093.760,245.292,424.197,177.189,19.362,152.706
C02583=1093.766,245.541,424.170,177.192,19.365,152.705
C02584=1093.772,245.789,424.143,177.195,19.366,152.705
C02585=1093.778,246.037,424.117,177.198,19.368,152.705
C02586=1093.783,246.286,424.090,177.201,19.370,152.705
C02587=1093.789,246.534,424.063,177.204,19.372,152.705
C02588=1093.794,246.783,424.036,177.207,19.374,152.705
C02589=1093.800,247.032,424.010,177.211,19.376,152.705
C02590=1093.806,247.280,423.984,177.213,19.377,152.705
C02591=1093.811,247.529,423.956,177.217,19.380,152.704
C02592=1093.816,247.777,423.930,177.220,19.382,152.704
C02593=1093.822,248.026,423.903,177.222,19.383,152.704
C02594=1093.827,248.274,423.876,177.226,19.386,152.704
C02595=1093.833,248.523,423.849,177.229,19.388,152.704
C02596=1093.838,248.771,423.822,177.232,19.389,152.704
C02597=1093.847,249.136,423.783,177.237,19.392,152.704
C02598=1093.855,249.501,423.743,177.241,19.395,152.704
C02599=1093.863,249.866,423.703,177.246,19.398,152.704
C02600=1093.871,250.231,423.663,177.250,19.401,152.703
C02601=1093.877,250.479,423.636,177.253,19.403,152.703
C02602=1093.882,250.728,423.609,177.256,19.405,152.703
C02603=1093.888,250.976,423.582,177.259,19.407,152.703
C02604=1093.893,251.225,423.555,177.262,19.409,152.703
C02605=1093.899,251.474,423.528,177.266,19.411,152.703
C02606=1093.904,251.722,423.500,177.268,19.413,152.703
C02607=1093.910,251.970,423.474,177.272,19.415,152.703
C02608=1093.915,252.219,423.446,177.275,19.417,152.703
C02609=1093.921,252.467,423.420,177.278,19.418,152.702
C02610=1093.926,252.716,423.392,177.281,19.421,152.702
C02611=1093.932,252.964,423.365,177.284,19.423,152.702
C02612=1093.938,253.213,423.338,177.288,19.425,152.702
C02613=1093.943,253.462,423.311,177.290,19.426,152.702
C02614=1093.949,253.710,423.283,177.293,19.429,152.702
C02615=1093.955,253.958,423.256,177.297,19.431,152.702
C02616=1093.960,254.207,423.229,177.299,19.432,152.702
C02617=1093.966,254.455,423.201,177.303,19.434,152.702
C02618=1093.971,254.704,423.174,177.306,19.437,152.701
C02619=1093.977,254.952,423.147,177.309,19.439,152.701
C02620=1093.982,255.200,423.119,177.312,19.440,152.701
C02621=1093.988,255.449,423.093,177.315,19.443,152.701
C02622=1093.994,255.698,423.065,177.319,19.445,152.701
C02623=1094.000,255.946,423.038,177.321,19.446,152.701
C02624=1094.005,256.194,423.010,177.324,19.448,152.701
C02625=1094.011,256.442,422.983,177.328,19.451,152.701
C02626=1094.017,256.691,422.956,177.331,19.453,152.701
C02627=1094.022,256.939,422.928,177.334,19.454,152.701
C02628=1094.028,257.188,422.901,177.337,19.456,152.700
C02629=1094.034,257.437,422.873,177.340,19.459,152.700
C02630=1094.040,257.685,422.846,177.344,19.461,152.700
C02631=1094.045,257.933,422.818,177.346,19.462,152.700
C02632=1094.050,258.182,422.791,177.350,19.464,152.700
C02633=1094.057,258.430,422.763,177.353,19.466,152.700
C02634=1094.062,258.679,422.736,177.355,19.468,152.700
C02635=1094.068,258.927,422.708,177.359,19.470,152.700
C02636=1094.074,259.175,422.680,177.362,19.472,152.699
C02637=1094.079,259.424,422.653,177.365,19.474,152.699
C02638=1094.085,259.672,422.625,177.368,19.476,152.699
C02639=1094.090,259.921,422.598,177.371,19.478,152.699
C02640=1094.096,260.169,422.570,177.375,19.480,152.699
C02641=1094.102,260.418,422.542,177.378,19.482,152.699
C02642=1094.107,260.666,422.515,177.380,19.484,152.699
C02643=1094.113,260.914,422.487,177.384,19.486,152.699
C02644=1094.119,261.163,422.459,177.387,19.488,152.699
C02645=1094.125,261.411,422.431,177.391,19.490,152.699
C02646=1094.130,261.659,422.404,177.393,19.492,152.699
C02647=1094.137,261.908,422.376,177.396,19.494,152.698
C02648=1094.142,262.156,422.348,177.400,19.496,152.698
C02649=1094.151,262.518,422.308,177.404,19.499,152.698
C02650=1094.159,262.881,422.267,177.409,19.502,152.698
C02651=1094.167,263.242,422.227,177.413,19.504,152.698
C02652=1094.176,263.605,422.186,177.418,19.508,152.698
C02653=1094.181,263.853,422.158,177.422,19.510,152.698
C02654=1094.188,264.101,422.131,177.424,19.511,152.697
C02655=1094.193,264.350,422.103,177.427,19.514,152.697
C02656=1094.199,264.598,422.074,177.431,19.516,152.697
C02657=1094.204,264.846,422.046,177.434,19.518,152.697
C02658=1094.210,265.094,422.018,177.437,19.520,152.697
C02659=1094.216,265.343,421.990,177.440,19.522,152.697
C02660=1094.221,265.592,421.963,177.443,19.524,152.697
C02661=1094.227,265.841,421.935,177.446,19.526,152.697
C02662=1094.232,266.089,421.907,177.450,19.529,152.697
C02663=1094.238,266.337,421.878,177.453,19.531,152.697
C02664=1094.243,266.585,421.850,177.456,19.532,152.697
C02665=1094.248,266.833,421.822,177.459,19.534,152.697
C02666=1094.254,267.082,421.794,177.462,19.537,152.697
C02667=1094.260,267.330,421.766,177.465,19.539,152.696
C02668=1094.266,267.578,421.737,177.469,19.541,152.696
C02669=1094.271,267.826,421.709,177.471,19.543,152.696
C02670=1094.277,268.075,421.681,177.475,19.545,152.696
C02671=1094.283,268.323,421.653,177.478,19.547,152.696
C02672=1094.289,268.572,421.624,177.481,19.549,152.696
C02673=1094.294,268.820,421.596,177.485,19.552,152.696
C02674=1094.300,269.069,421.568,177.487,19.554,152.696
C02675=1094.305,269.317,421.540,177.490,19.556,152.696
C02676=1094.311,269.566,421.512,177.494,19.558,152.696
C02677=1094.317,269.813,421.483,177.497,19.560,152.696
C02678=1094.323,270.062,421.455,177.500,19.562,152.696
C02679=1094.328,270.310,421.427,177.503,19.564,152.695
C02680=1094.334,270.559,421.399,177.506,19.566,152.696
C02681=1094.340,270.806,421.370,177.509,19.569,152.695
C02682=1094.345,271.055,421.341,177.512,19.571,152.695
C02683=1094.351,271.304,421.313,177.516,19.573,152.695
C02684=1094.356,271.552,421.285,177.519,19.575,152.695
C02685=1094.362,271.800,421.256,177.521,19.577,152.695
C02686=1094.368,272.048,421.228,177.525,19.579,152.695
C02687=1094.374,272.297,421.199,177.528,19.581,152.695
C02688=1094.379,272.544,421.171,177.531,19.584,152.695
C02689=1094.385,272.793,421.142,177.535,19.586,152.695
C02690=1094.390,273.041,421.114,177.538,19.588,152.695
C02691=1094.396,273.289,421.085,177.540,19.590,152.695
C02692=1094.402,273.538,421.056,177.544,19.592,152.695
C02693=1094.407,273.786,421.029,177.547,19.594,152.695
C02694=1094.413,274.035,420.999,177.550,19.597,152.695
C02695=1094.418,274.283,420.971,177.554,19.599,152.695
C02696=1094.425,274.531,420.942,177.557,19.601,152.694
C02697=1094.430,274.780,420.913,177.559,19.603,152.695
C02698=1094.435,275.027,420.884,177.562,19.605,152.694
C02699=1094.441,275.276,420.856,177.566,19.608,152.694
C02700=1094.447,275.524,420.827,177.569,19.610,152.694
C02701=1094.455,275.890,420.785,177.574,19.613,152.694
C02702=1094.463,276.254,420.743,177.578,19.616,152.694
C02703=1094.472,276.619,420.700,177.583,19.620,152.694
C02704=1094.480,276.984,420.658,177.588,19.623,152.694
C02705=1094.486,277.232,420.629,177.591,19.626,152.694
C02706=1094.491,277.480,420.601,177.593,19.627,152.694
C02707=1094.497,277.729,420.571,177.597,19.629,152.694
C02708=1094.503,277.977,420.542,177.600,19.632,152.694
C02709=1094.508,278.225,420.514,177.603,19.634,152.694
C02710=1094.514,278.473,420.484,177.607,19.636,152.694
C02711=1094.520,278.721,420.455,177.610,19.639,152.694
C02712=1094.525,278.970,420.426,177.613,19.641,152.694
C02713=1094.531,279.218,420.398,177.616,19.643,152.694
C02714=1094.537,279.466,420.369,177.619,19.645,152.694
C02715=1094.542,279.715,420.340,177.622,19.647,152.694
C02716=1094.548,279.962,420.311,177.625,19.649,152.693
C02717=1094.553,280.211,420.282,177.628,19.652,152.693
C02718=1094.560,280.459,420.252,177.632,19.654,152.693
C02719=1094.565,280.708,420.224,177.635,19.657,152.693
C02720=1094.570,280.955,420.195,177.638,19.659,152.693
C02721=1094.576,281.204,420.165,177.642,19.661,152.693
C02722=1094.582,281.452,420.136,177.645,19.664,152.693
C02723=1094.588,281.700,420.107,177.648,19.666,152.693
C02724=1094.593,281.948,420.078,177.650,19.668,152.693
C02725=1094.599,282.197,420.049,177.654,19.670,152.693
C02726=1094.604,282.445,420.019,177.657,19.673,152.693
C02727=1094.610,282.693,419.991,177.660,19.675,152.693
C02728=1094.615,282.941,419.961,177.663,19.677,152.693
C02729=1094.621,283.190,419.931,177.666,19.680,152.693
C02730=1094.627,283.438,419.902,177.670,19.682,152.693
C02731=1094.632,283.686,419.873,177.673,19.684,152.693
C02732=1094.638,283.934,419.844,177.676,19.687,152.693
C02733=1094.644,284.182,419.814,177.679,19.689,152.693
C02734=1094.649,284.431,419.785,177.682,19.692,152.693
C02735=1094.655,284.679,419.756,177.685,19.693,152.693
C02736=1094.660,284.926,419.726,177.688,19.696,152.693
C02737=1094.666,285.175,419.697,177.691,19.698,152.693
C02738=1094.672,285.423,419.668,177.695,19.701,152.693
C02739=1094.678,285.671,419.638,177.698,19.703,152.693
C02740=1094.683,285.920,419.609,177.701,19.705,152.693
C02741=1094.688,286.168,419.579,177.704,19.708,152.693
C02742=1094.695,286.415,419.549,177.707,19.710,152.693
C02743=1094.700,286.664,419.520,177.711,19.712,152.693
C02744=1094.706,286.912,419.490,177.714,19.715,152.693
C02745=1094.712,287.160,419.461,177.717,19.717,152.693
C02746=1094.717,287.409,419.432,177.720,19.720,152.693
C02747=1094.723,287.657,419.402,177.724,19.722,152.693
C02748=1094.728,287.906,419.372,177.727,19.724,152.693
C02749=1094.734,288.152,419.343,177.730,19.727,152.693
C02750=1094.740,288.401,419.313,177.732,19.729,152.693
C02751=1094.745,288.649,419.284,177.735,19.731,152.693
C02752=1094.751,288.898,419.254,177.739,19.733,152.693
C02753=1094.760,289.272,419.209,177.744,19.737,152.693
C02754=1094.769,289.646,419.165,177.748,19.741,152.693
C02755=1094.777,290.020,419.119,177.753,19.744,152.693
C02756=1094.785,290.394,419.074,177.758,19.748,152.693
C02757=1094.792,290.643,419.045,177.761,19.751,152.693
C02758=1094.798,290.890,419.015,177.764,19.753,152.693
C02759=1094.803,291.139,418.985,177.768,19.755,152.693
C02760=1094.809,291.387,418.956,177.771,19.758,152.693
C02761=1094.814,291.635,418.925,177.774,19.760,152.693
C02762=1094.819,291.883,418.896,177.777,19.763,152.693
C02763=1094.825,292.131,418.866,177.780,19.765,152.693
C02764=1094.831,292.379,418.836,177.784,19.768,152.693
C02765=1094.836,292.627,418.806,177.787,19.770,152.693
C02766=1094.842,292.875,418.776,177.790,19.773,152.693
C02767=1094.848,293.123,418.746,177.793,19.775,152.693
C02768=1094.853,293.372,418.716,177.796,19.778,152.693
C02769=1094.859,293.620,418.686,177.799,19.780,152.693
C02770=1094.865,293.868,418.656,177.802,19.783,152.693
C02771=1094.870,294.116,418.626,177.806,19.785,152.693
C02772=1094.876,294.364,418.596,177.809,19.787,152.693
C02773=1094.882,294.612,418.566,177.812,19.790,152.693
C02774=1094.888,294.860,418.535,177.815,19.793,152.693
C02775=1094.893,295.108,418.506,177.818,19.795,152.693
C02776=1094.899,295.356,418.475,177.822,19.797,152.693
C02777=1094.905,295.604,418.445,177.825,19.800,152.693
C02778=1094.910,295.852,418.415,177.828,19.803,152.693
C02779=1094.916,296.100,418.385,177.831,19.805,152.693
C02780=1094.922,296.348,418.355,177.834,19.807,152.693
C02781=1094.927,296.596,418.325,177.837,19.810,152.693
C02782=1094.933,296.844,418.295,177.840,19.813,152.693
C02783=1094.938,297.092,418.264,177.844,19.815,152.693
C02784=1094.944,297.342,418.234,177.847,19.818,152.693
C02785=1094.950,297.589,418.203,177.850,19.820,152.693
C02786=1094.956,297.837,418.173,177.853,19.823,152.694
C02787=1094.962,298.085,418.143,177.856,19.825,152.693
C02788=1094.968,298.333,418.112,177.859,19.828,152.694
C02789=1094.972,298.582,418.082,177.862,19.830,152.694
C02790=1094.978,298.829,418.052,177.866,19.833,152.694
C02791=1094.984,299.077,418.021,177.869,19.836,152.694
C02792=1094.989,299.325,417.990,177.872,19.838,152.694
C02793=1094.995,299.573,417.960,177.875,19.841,152.694
C02794=1095.001,299.821,417.930,177.878,19.844,152.694
C02795=1095.006,300.069,417.899,177.882,19.847,152.694
C02796=1095.011,300.318,417.869,177.885,19.849,152.694
C02797=1095.017,300.565,417.839,177.888,19.852,152.694
C02798=1095.022,300.814,417.808,177.891,19.855,152.694
C02799=1095.028,301.061,417.777,177.894,19.857,152.694
C02800=1095.033,301.310,417.747,177.897,19.860,152.694
C02801=1095.039,301.557,417.716,177.900,19.862,152.694
C02802=1095.045,301.806,417.685,177.903,19.865,152.694
C02803=1095.050,302.054,417.655,177.907,19.868,152.695
C02804=1095.056,302.302,417.624,177.910,19.870,152.695
C02805=1095.065,302.690,417.576,177.915,19.875,152.695
C02806=1095.074,303.078,417.528,177.920,19.879,152.695
C02807=1095.082,303.466,417.480,177.924,19.883,152.695
C02808=1095.091,303.854,417.432,177.930,19.887,152.695
C02809=1095.097,304.102,417.401,177.933,19.890,152.695
C02810=1095.103,304.350,417.370,177.936,19.893,152.695
C02811=1095.108,304.598,417.339,177.939,19.896,152.695
C02812=1095.113,304.846,417.308,177.942,19.898,152.695
C02813=1095.119,305.094,417.278,177.945,19.901,152.696
C02814=1095.125,305.342,417.246,177.948,19.903,152.696
C02815=1095.131,305.590,417.216,177.951,19.906,152.696
C02816=1095.136,305.838,417.185,177.954,19.909,152.696
C02817=1095.142,306.086,417.154,177.958,19.912,152.696
C02818=1095.147,306.333,417.123,177.961,19.915,152.696
C02819=1095.154,306.582,417.092,177.964,19.917,152.696
C02820=1095.159,306.830,417.061,177.967,19.920,152.696
C02821=1095.165,307.078,417.031,177.971,19.923,152.696
C02822=1095.170,307.325,416.999,177.974,19.925,152.696
C02823=1095.176,307.574,416.968,177.977,19.928,152.696
C02824=1095.182,307.821,416.937,177.980,19.931,152.696
C02825=1095.188,308.069,416.906,177.983,19.933,152.697
C02826=1095.193,308.318,416.875,177.987,19.937,152.697
C02827=1095.199,308.565,416.844,177.990,19.939,152.697
C02828=1095.205,308.813,416.813,177.993,19.942,152.697
C02829=1095.211,309.062,416.781,177.996,19.945,152.697
C02830=1095.216,309.310,416.751,177.999,19.947,152.697
C02831=1095.221,309.558,416.720,178.002,19.950,152.697
C02832=1095.228,309.806,416.688,178.005,19.953,152.697
C02833=1095.233,310.054,416.657,178.008,19.956,152.697
C02834=1095.239,310.301,416.626,178.012,19.959,152.697
C02835=1095.245,310.550,416.595,178.015,19.961,152.697
C02836=1095.250,310.797,416.563,178.018,19.964,152.698
C02837=1095.257,311.044,416.532,178.021,19.967,152.698
C02838=1095.262,311.293,416.501,178.024,19.970,152.698
C02839=1095.268,311.541,416.469,178.027,19.972,152.698
C02840=1095.274,311.789,416.438,178.030,19.975,152.698
C02841=1095.279,312.037,416.407,178.033,19.978,152.698
C02842=1095.285,312.285,416.376,178.037,19.981,152.698
C02843=1095.291,312.533,416.344,178.040,19.984,152.698
C02844=1095.297,312.780,416.313,178.043,19.987,152.698
C02845=1095.303,313.029,416.282,178.046,19.989,152.699
C02846=1095.308,313.276,416.250,178.050,19.992,152.699
C02847=1095.314,313.525,416.218,178.052,19.995,152.699
C02848=1095.319,313.773,416.187,178.056,19.997,152.699
C02849=1095.326,314.021,416.156,178.060,20.001,152.699
C02850=1095.332,314.268,416.124,178.062,20.004,152.699
C02851=1095.338,314.516,416.092,178.066,20.006,152.699
C02852=1095.343,314.764,416.062,178.068,20.009,152.699
C02853=1095.349,315.012,416.030,178.072,20.012,152.699
C02854=1095.355,315.260,415.998,178.075,20.014,152.700
C02855=1095.361,315.508,415.966,178.078,20.018,152.700
C02856=1095.366,315.756,415.935,178.081,20.021,152.700
C02857=1095.375,316.147,415.884,178.086,20.025,152.700
C02858=1095.384,316.538,415.835,178.091,20.030,152.700
C02859=1095.392,316.928,415.785,178.096,20.035,152.701
C02860=1095.401,317.319,415.734,178.101,20.039,152.701
C02861=1095.407,317.567,415.702,178.104,20.042,152.701
C02862=1095.412,317.815,415.671,178.107,20.046,152.701
C02863=1095.418,318.062,415.639,178.110,20.049,152.702
C02864=1095.423,318.311,415.608,178.113,20.052,152.702
C02865=1095.429,318.559,415.576,178.116,20.055,152.702
C02866=1095.435,318.807,415.544,178.119,20.058,152.702
C02867=1095.440,319.054,415.512,178.123,20.061,152.702
C02868=1095.446,319.303,415.480,178.126,20.064,152.702
C02869=1095.452,319.549,415.448,178.129,20.067,152.702
C02870=1095.457,319.798,415.415,178.132,20.070,152.703
C02871=1095.463,320.046,415.383,178.135,20.073,152.703
C02872=1095.468,320.294,415.352,178.138,20.077,152.703
C02873=1095.474,320.542,415.320,178.141,20.080,152.703
C02874=1095.480,320.789,415.288,178.144,20.082,152.703
C02875=1095.486,321.038,415.256,178.147,20.085,152.704
C02876=1095.491,321.285,415.224,178.151,20.089,152.704
C02877=1095.496,321.534,415.192,178.154,20.092,152.704
C02878=1095.502,321.781,415.160,178.157,20.095,152.704
C02879=1095.508,322.029,415.127,178.160,20.098,152.704
C02880=1095.514,322.277,415.095,178.163,20.101,152.704
C02881=1095.519,322.524,415.063,178.167,20.104,152.705
C02882=1095.525,322.773,415.031,178.169,20.107,152.705
C02883=1095.531,323.021,414.998,178.172,20.110,152.705
C02884=1095.536,323.268,414.966,178.175,20.113,152.705
C02885=1095.542,323.516,414.934,178.179,20.117,152.706
C02886=1095.548,323.764,414.903,178.182,20.120,152.706
C02887=1095.553,324.012,414.869,178.185,20.123,152.706
C02888=1095.559,324.260,414.837,178.188,20.126,152.706
C02889=1095.565,324.507,414.806,178.191,20.129,152.706
C02890=1095.571,324.755,414.773,178.194,20.132,152.707
C02891=1095.576,325.004,414.740,178.197,20.135,152.707
C02892=1095.582,325.252,414.708,178.201,20.139,152.707
C02893=1095.588,325.499,414.676,178.204,20.142,152.707
C02894=1095.594,325.747,414.644,178.207,20.145,152.707
C02895=1095.599,325.995,414.611,178.210,20.148,152.708
C02896=1095.605,326.242,414.579,178.213,20.152,152.708
C02897=1095.611,326.490,414.546,178.216,20.155,152.708
C02898=1095.617,326.738,414.514,178.219,20.158,152.708
C02899=1095.622,326.987,414.482,178.222,20.161,152.708
C02900=1095.628,327.234,414.449,178.226,20.164,152.709
C02901=1095.634,327.482,414.417,178.229,20.167,152.709
C02902=1095.640,327.730,414.384,178.232,20.170,152.709
C02903=1095.646,327.977,414.351,178.235,20.174,152.709
C02904=1095.652,328.225,414.319,178.238,20.177,152.710
C02905=1095.657,328.473,414.286,178.241,20.180,152.710
C02906=1095.663,328.721,414.254,178.244,20.183,152.710
C02907=1095.669,328.968,414.221,178.248,20.187,152.710
C02908=1095.675,329.216,414.188,178.251,20.190,152.710
C02909=1095.684,329.600,414.138,178.256,20.195,152.711
C02910=1095.693,329.984,414.087,178.260,20.200,152.711
C02911=1095.701,330.368,414.036,178.265,20.205,152.711
C02912=1095.711,330.751,413.986,178.270,20.210,152.712
C02913=1095.716,330.999,413.953,178.273,20.213,152.712
C02914=1095.722,331.247,413.920,178.276,20.216,152.712
C02915=1095.728,331.495,413.888,178.280,20.220,152.713
C02916=1095.734,331.743,413.855,178.282,20.223,152.713
C02917=1095.740,331.991,413.822,178.285,20.226,152.713
C02918=1095.746,332.239,413.789,178.289,20.230,152.713
C02919=1095.752,332.486,413.756,178.292,20.233,152.714
C02920=1095.757,332.734,413.724,178.295,20.237,152.714
C02921=1095.762,332.982,413.691,178.298,20.240,152.714
C02922=1095.769,333.229,413.658,178.301,20.244,152.715
C02923=1095.774,333.477,413.624,178.305,20.247,152.715
C02924=1095.780,333.725,413.591,178.307,20.251,152.715
C02925=1095.786,333.973,413.558,178.310,20.254,152.715
C02926=1095.792,334.221,413.525,178.314,20.258,152.716
C02927=1095.797,334.468,413.492,178.317,20.261,152.716
C02928=1095.803,334.716,413.459,178.319,20.264,152.716
C02929=1095.808,334.963,413.426,178.323,20.268,152.716
C02930=1095.814,335.211,413.393,178.326,20.271,152.717
C02931=1095.820,335.459,413.360,178.329,20.275,152.717
C02932=1095.826,335.707,413.327,178.332,20.278,152.717
C02933=1095.831,335.955,413.293,178.335,20.282,152.718
C02934=1095.837,336.203,413.260,178.338,20.285,152.718
C02935=1095.843,336.450,413.227,178.341,20.289,152.718
C02936=1095.849,336.698,413.194,178.345,20.292,152.718
C02937=1095.854,336.946,413.160,178.348,20.296,152.719
C02938=1095.860,337.194,413.127,178.350,20.299,152.719
C02939=1095.866,337.442,413.094,178.354,20.303,152.719
C02940=1095.872,337.689,413.061,178.357,20.306,152.720
C02941=1095.878,337.937,413.027,178.360,20.310,152.720
C02942=1095.883,338.185,412.994,178.363,20.313,152.720
C02943=1095.889,338.432,412.961,178.366,20.317,152.721
C02944=1095.895,338.680,412.928,178.369,20.321,152.721
C02945=1095.900,338.928,412.894,178.372,20.324,152.721
C02946=1095.906,339.175,412.860,178.376,20.328,152.722
C02947=1095.912,339.423,412.827,178.378,20.331,152.722
C02948=1095.917,339.671,412.794,178.382,20.335,152.722
C02949=1095.923,339.919,412.760,178.385,20.339,152.723
C02950=1095.929,340.166,412.726,178.388,20.343,152.723
C02951=1095.934,340.414,412.693,178.391,20.346,152.723
C02952=1095.940,340.662,412.659,178.393,20.350,152.724
C02953=1095.946,340.909,412.625,178.397,20.354,152.724
C02954=1095.951,341.157,412.592,178.400,20.357,152.724
C02955=1095.958,341.405,412.559,178.403,20.361,152.725
C02956=1095.964,341.652,412.525,178.406,20.364,152.725
C02957=1095.969,341.900,412.492,178.410,20.368,152.725
C02958=1095.975,342.147,412.458,178.412,20.371,152.726
C02959=1095.981,342.395,412.425,178.416,20.375,152.726
C02960=1095.986,342.643,412.390,178.419,20.379,152.726
C02961=1095.995,343.021,412.339,178.423,20.385,152.727
C02962=1096.003,343.399,412.288,178.428,20.391,152.728
C02963=1096.012,343.776,412.236,178.433,20.396,152.728
C02964=1096.021,344.154,412.185,178.438,20.402,152.729
C02965=1096.027,344.402,412.151,178.440,20.406,152.729
C02966=1096.033,344.649,412.117,178.443,20.409,152.729
C02967=1096.039,344.898,412.083,178.447,20.413,152.730
C02968=1096.045,345.145,412.049,178.450,20.418,152.730
C02969=1096.050,345.393,412.016,178.453,20.421,152.731
C02970=1096.055,345.640,411.981,178.456,20.425,152.731
C02971=1096.061,345.888,411.947,178.459,20.428,152.731
C02972=1096.067,346.135,411.914,178.462,20.433,152.732
C02973=1096.073,346.383,411.880,178.465,20.436,152.732
C02974=1096.078,346.630,411.846,178.468,20.440,152.733
C02975=1096.085,346.878,411.811,178.471,20.444,152.733
C02976=1096.090,347.126,411.777,178.474,20.448,152.733
C02977=1096.096,347.374,411.743,178.477,20.452,152.734
C02978=1096.101,347.621,411.709,178.480,20.456,152.734
C02979=1096.107,347.868,411.675,178.483,20.460,152.735
C02980=1096.112,348.116,411.641,178.486,20.464,152.735
C02981=1096.119,348.364,411.607,178.489,20.467,152.736
C02982=1096.124,348.612,411.573,178.492,20.472,152.736
C02983=1096.130,348.859,411.539,178.496,20.476,152.736
C02984=1096.135,349.106,411.504,178.498,20.480,152.737
C02985=1096.142,349.354,411.470,178.502,20.484,152.737
C02986=1096.148,349.602,411.436,178.504,20.488,152.738
C02987=1096.153,349.849,411.401,178.508,20.492,152.738
C02988=1096.159,350.097,411.367,178.510,20.496,152.739
C02989=1096.165,350.344,411.333,178.514,20.499,152.739
C02990=1096.170,350.592,411.298,178.516,20.503,152.740
C02991=1096.176,350.839,411.264,178.520,20.508,152.740
C02992=1096.182,351.087,411.230,178.523,20.512,152.740
C02993=1096.187,351.334,411.195,178.526,20.516,152.741
C02994=1096.194,351.582,411.161,178.529,20.520,152.741
C02995=1096.200,351.830,411.127,178.532,20.524,152.742
C02996=1096.205,352.077,411.092,178.535,20.528,152.742
C02997=1096.211,352.325,411.058,178.538,20.532,152.743
C02998=1096.216,352.573,411.023,178.541,20.536,152.743
C02999=1096.222,352.820,410.989,178.544,20.540,152.744
C03000=1096.228,353.067,410.955,178.547,20.544,152.744
C03001=1096.234,353.316,410.920,178.550,20.549,152.745
C03002=1096.240,353.562,410.885,178.554,20.553,152.745
C03003=1096.245,353.810,410.850,178.556,20.556,152.745
C03004=1096.251,354.058,410.816,178.560,20.561,152.746
C03005=1096.257,354.305,410.781,178.563,20.565,152.746
C03006=1096.262,354.553,410.747,178.565,20.569,152.747
C03007=1096.268,354.800,410.712,178.569,20.574,152.747
C03008=1096.274,355.048,410.677,178.571,20.577,152.748
C03009=1096.279,355.295,410.643,178.574,20.582,152.749
C03010=1096.285,355.543,410.607,178.578,20.586,152.749
C03011=1096.291,355.790,410.573,178.580,20.590,152.750
C03012=1096.296,356.038,410.538,178.584,20.595,152.750
C03013=1096.306,356.418,410.485,178.588,20.601,152.751
C03014=1096.315,356.798,410.432,178.593,20.608,152.752
C03015=1096.323,357.178,410.377,178.597,20.614,152.752
C03016=1096.332,357.558,410.324,178.602,20.621,152.753
C03017=1096.338,357.806,410.289,178.605,20.625,152.754
C03018=1096.344,358.053,410.255,178.608,20.630,152.754
C03019=1096.350,358.302,410.220,178.611,20.634,152.755
C03020=1096.355,358.549,410.184,178.614,20.638,152.755
C03021=1096.362,358.796,410.149,178.617,20.643,152.756
C03022=1096.367,359.044,410.114,178.620,20.647,152.756
C03023=1096.372,359.290,410.079,178.623,20.651,152.757
C03024=1096.379,359.538,410.045,178.626,20.656,152.758
C03025=1096.384,359.785,410.009,178.629,20.660,152.758
C03026=1096.390,360.034,409.974,178.632,20.664,152.759
C03027=1096.396,360.280,409.940,178.635,20.669,152.759
C03028=1096.402,360.528,409.904,178.638,20.673,152.760
C03029=1096.407,360.776,409.869,178.641,20.678,152.760
C03030=1096.413,361.023,409.833,178.644,20.682,152.761
C03031=1096.419,361.270,409.798,178.647,20.687,152.762
C03032=1096.425,361.518,409.764,178.650,20.691,152.762
C03033=1096.431,361.765,409.728,178.653,20.696,152.763
C03034=1096.436,362.012,409.693,178.656,20.700,152.763
C03035=1096.442,362.260,409.657,178.659,20.705,152.764
C03036=1096.447,362.508,409.623,178.662,20.710,152.764
C03037=1096.453,362.755,409.587,178.665,20.714,152.765
C03038=1096.460,363.002,409.552,178.668,20.719,152.766
C03039=1096.466,363.250,409.516,178.671,20.723,152.766
C03040=1096.472,363.497,409.481,178.674,20.728,152.767
C03041=1096.477,363.744,409.445,178.676,20.732,152.767
C03042=1096.483,363.992,409.409,178.680,20.737,152.768
C03043=1096.488,364.239,409.375,178.683,20.741,152.769
C03044=1096.494,364.487,409.339,178.686,20.746,152.769
C03045=1096.500,364.734,409.304,178.688,20.750,152.770
C03046=1096.506,364.981,409.269,178.691,20.755,152.771
C03047=1096.512,365.228,409.233,178.695,20.760,152.771
C03048=1096.518,365.476,409.198,178.698,20.765,152.772
C03049=1096.524,365.724,409.162,178.701,20.770,152.772
C03050=1096.529,365.971,409.126,178.703,20.774,152.773
C03051=1096.535,366.218,409.091,178.706,20.779,152.774
C03052=1096.541,366.465,409.055,178.709,20.784,152.774
C03053=1096.546,366.713,409.019,178.712,20.789,152.775
C03054=1096.551,366.960,408.984,178.716,20.793,152.776
C03055=1096.558,367.207,408.947,178.718,20.798,152.776
C03056=1096.563,367.454,408.912,178.721,20.803,152.777
C03057=1096.569,367.702,408.876,178.724,20.807,152.778
C03058=1096.575,367.950,408.840,178.727,20.813,152.778
C03059=1096.581,368.197,408.805,178.730,20.817,152.779
C03060=1096.587,368.444,408.769,178.732,20.822,152.780
C03061=1096.592,368.691,408.733,178.736,20.827,152.780
C03062=1096.598,368.939,408.697,178.739,20.832,152.781
C03063=1096.604,369.186,408.661,178.742,20.837,152.782
C03064=1096.609,369.433,408.626,178.745,20.841,152.782
C03065=1096.619,369.829,408.568,178.749,20.849,152.784
C03066=1096.628,370.224,408.511,178.754,20.857,152.785
C03067=1096.637,370.619,408.453,178.759,20.865,152.786
C03068=1096.647,371.014,408.396,178.763,20.873,152.787
C03069=1096.652,371.262,408.360,178.766,20.878,152.788
C03070=1096.659,371.509,408.323,178.769,20.883,152.788
C03071=1096.664,371.756,408.288,178.772,20.888,152.789
C03072=1096.670,372.003,408.251,178.775,20.893,152.790
C03073=1096.676,372.251,408.215,178.778,20.898,152.791
C03074=1096.682,372.499,408.179,178.781,20.903,152.791
C03075=1096.687,372.745,408.143,178.784,20.908,152.792
C03076=1096.693,372.993,408.108,178.787,20.913,152.793
C03077=1096.700,373.240,408.071,178.790,20.918,152.794
C03078=1096.705,373.487,408.034,178.792,20.923,152.794
C03079=1096.711,373.734,407.999,178.795,20.928,152.795
C03080=1096.717,373.981,407.962,178.798,20.933,152.796
C03081=1096.722,374.229,407.926,178.801,20.938,152.797
C03082=1096.729,374.476,407.890,178.804,20.943,152.797
C03083=1096.734,374.723,407.853,178.807,20.949,152.798
C03084=1096.740,374.971,407.817,178.810,20.954,152.799
C03085=1096.746,375.218,407.781,178.813,20.959,152.800
C03086=1096.752,375.465,407.744,178.815,20.964,152.800
C03087=1096.757,375.712,407.708,178.818,20.970,152.801
C03088=1096.763,375.960,407.671,178.821,20.975,152.802
C03089=1096.769,376.207,407.635,178.824,20.981,152.803
C03090=1096.775,376.454,407.598,178.827,20.986,152.804
C03091=1096.780,376.701,407.562,178.830,20.991,152.805
C03092=1096.786,376.948,407.525,178.832,20.996,152.805
C03093=1096.792,377.195,407.489,178.835,21.001,152.806
C03094=1096.798,377.443,407.452,178.838,21.007,152.807
C03095=1096.804,377.690,407.415,178.841,21.012,152.808
C03096=1096.809,377.937,407.379,178.844,21.017,152.809
C03097=1096.815,378.184,407.343,178.846,21.023,152.810
C03098=1096.821,378.431,407.306,178.849,21.028,152.810
C03099=1096.827,378.679,407.270,178.852,21.034,152.811
C03100=1096.832,378.926,407.232,178.855,21.039,152.812
C03101=1096.839,379.173,407.196,178.858,21.044,152.813
C03102=1096.844,379.420,407.159,178.861,21.050,152.814
C03103=1096.850,379.667,407.123,178.864,21.055,152.815
C03104=1096.856,379.914,407.086,178.866,21.061,152.815
C03105=1096.861,380.161,407.049,178.869,21.066,152.816
C03106=1096.868,380.408,407.012,178.872,21.072,152.817
C03107=1096.873,380.656,406.975,178.875,21.077,152.818
C03108=1096.880,380.903,406.939,178.878,21.083,152.819
C03109=1096.885,381.150,406.902,178.880,21.088,152.820
C03110=1096.891,381.398,406.865,178.883,21.094,152.821
C03111=1096.897,381.644,406.828,178.886,21.099,152.822
C03112=1096.903,381.891,406.791,178.889,21.105,152.822
C03113=1096.909,382.139,406.754,178.892,21.110,152.823
C03114=1096.915,382.386,406.717,178.894,21.116,152.824
C03115=1096.921,382.633,406.680,178.898,21.122,152.825
C03116=1096.926,382.881,406.643,178.901,21.128,152.826
C03117=1096.934,383.181,406.598,178.904,21.135,152.827
C03118=1096.942,383.528,406.546,178.908,21.143,152.829
C03119=1096.949,383.875,406.493,178.912,21.151,152.830
C03120=1096.958,384.222,406.442,178.916,21.159,152.831
C03121=1096.966,384.570,406.389,178.919,21.167,152.833
C03122=1096.971,384.817,406.352,178.922,21.172,152.833
C03123=1096.977,385.064,406.315,178.926,21.179,152.834
C03124=1096.983,385.311,406.277,178.928,21.185,152.835
C03125=1096.989,385.558,406.240,178.931,21.190,152.836
C03126=1096.995,385.805,406.203,178.934,21.196,152.837
C03127=1097.001,386.052,406.166,178.936,21.202,152.838
C03128=1097.007,386.299,406.128,178.939,21.208,152.839
C03129=1097.012,386.546,406.091,178.942,21.214,152.840
C03130=1097.018,386.793,406.054,178.944,21.219,152.841
C03131=1097.024,387.040,406.017,178.948,21.226,152.842
C03132=1097.030,387.287,405.979,178.950,21.232,152.843
C03133=1097.035,387.535,405.942,178.953,21.238,152.844
C03134=1097.041,387.781,405.904,178.956,21.244,152.845
C03135=1097.047,388.029,405.867,178.959,21.249,152.846
C03136=1097.053,388.275,405.829,178.961,21.255,152.847
C03137=1097.059,388.523,405.791,178.965,21.262,152.848
C03138=1097.065,388.770,405.754,178.967,21.268,152.849
C03139=1097.071,389.017,405.716,178.970,21.274,152.850
C03140=1097.077,389.264,405.678,178.972,21.280,152.851
C03141=1097.082,389.511,405.641,178.975,21.286,152.853
C03142=1097.088,389.758,405.604,178.978,21.292,152.854
C03143=1097.094,390.005,405.566,178.981,21.299,152.855
C03144=1097.100,390.251,405.528,178.984,21.304,152.856
C03145=1097.106,390.499,405.491,178.986,21.310,152.857
C03146=1097.112,390.746,405.453,178.989,21.316,152.858
C03147=1097.118,390.993,405.415,178.991,21.322,152.859
C03148=1097.124,391.240,405.378,178.995,21.329,152.860
C03149=1097.130,391.486,405.340,178.997,21.336,152.861
C03150=1097.136,391.733,405.302,179.000,21.342,152.862
C03151=1097.142,391.981,405.265,179.002,21.348,152.863
C03152=1097.148,392.228,405.227,179.006,21.354,152.864
C03153=1097.154,392.475,405.189,179.008,21.360,152.865
C03154=1097.160,392.721,405.151,179.011,21.367,152.867
C03155=1097.165,392.968,405.113,179.013,21.373,152.868
C03156=1097.171,393.216,405.075,179.017,21.380,152.869
C03157=1097.177,393.463,405.037,179.019,21.386,152.870
C03158=1097.183,393.709,404.999,179.022,21.392,152.871
C03159=1097.188,393.956,404.961,179.024,21.398,152.872
C03160=1097.195,394.204,404.923,179.027,21.405,152.873
C03161=1097.201,394.451,404.885,179.030,21.412,152.875
C03162=1097.207,394.697,404.847,179.032,21.418,152.876
C03163=1097.212,394.944,404.809,179.035,21.425,152.877
C03164=1097.218,395.192,404.771,179.038,21.432,152.878
C03165=1097.224,395.438,404.732,179.041,21.438,152.879
C03166=1097.230,395.685,404.694,179.043,21.444,152.880
C03167=1097.236,395.932,404.656,179.046,21.451,152.881
C03168=1097.242,396.179,404.618,179.049,21.458,152.883
C03169=1097.247,396.426,404.580,179.051,21.464,152.884
C03170=1097.252,396.644,404.546,179.054,21.470,152.885
C03171=1097.258,396.861,404.512,179.056,21.476,152.886
C03172=1097.263,397.079,404.478,179.058,21.482,152.887
C03173=1097.268,397.297,404.444,179.061,21.488,152.888
C03174=1097.273,397.514,404.411,179.063,21.494,152.889
C03175=1097.278,397.732,404.377,179.065,21.500,152.890
C03176=1097.284,397.949,404.343,179.067,21.506,152.891
C03177=1097.289,398.167,404.309,179.070,21.512,152.893
C03178=1097.295,398.414,404.271,179.072,21.518,152.894
C03179=1097.301,398.661,404.233,179.076,21.526,152.895
C03180=1097.306,398.908,404.194,179.078,21.532,152.896
C03181=1097.313,399.155,404.156,179.080,21.539,152.898
C03182=1097.318,399.401,404.117,179.083,21.546,152.899
C03183=1097.325,399.649,404.079,179.086,21.553,152.900
C03184=1097.330,399.895,404.040,179.088,21.559,152.901
C03185=1097.336,400.143,404.001,179.091,21.567,152.903
C03186=1097.342,400.390,403.963,179.094,21.573,152.904
C03187=1097.348,400.636,403.924,179.097,21.581,152.905
C03188=1097.354,400.884,403.886,179.099,21.588,152.907
C03189=1097.360,401.130,403.847,179.102,21.595,152.908
C03190=1097.366,401.377,403.808,179.104,21.602,152.909
C03191=1097.371,401.624,403.770,179.106,21.609,152.911
C03192=1097.378,401.871,403.731,179.109,21.616,152.912
C03193=1097.383,402.118,403.692,179.112,21.623,152.913
C03194=1097.390,402.365,403.653,179.115,21.631,152.915
C03195=1097.395,402.612,403.614,179.117,21.637,152.916
C03196=1097.401,402.859,403.576,179.120,21.645,152.917
C03197=1097.407,403.105,403.537,179.122,21.652,152.919
C03198=1097.413,403.353,403.498,179.125,21.659,152.920
C03199=1097.418,403.600,403.459,179.128,21.666,152.921
C03200=1097.425,403.846,403.421,179.130,21.674,152.923
C03201=1097.431,404.093,403.381,179.133,21.681,152.924
C03202=1097.437,404.340,403.342,179.136,21.688,152.925
C03203=1097.442,404.586,403.303,179.138,21.695,152.927
C03204=1097.448,404.834,403.264,179.141,21.703,152.928
C03205=1097.455,405.081,403.225,179.143,21.710,152.930
C03206=1097.460,405.327,403.186,179.146,21.718,152.931
C03207=1097.466,405.575,403.147,179.149,21.725,152.933
C03208=1097.472,405.821,403.108,179.151,21.733,152.934
C03209=1097.478,406.068,403.068,179.154,21.741,152.936
C03210=1097.483,406.315,403.029,179.156,21.748,152.937
C03211=1097.490,406.561,402.991,179.159,21.755,152.938
C03212=1097.496,406.809,402.951,179.161,21.763,152.940
C03213=1097.502,407.055,402.912,179.164,21.770,152.941
C03214=1097.508,407.302,402.873,179.167,21.778,152.943
C03215=1097.514,407.549,402.833,179.169,21.786,152.944
C03216=1097.519,407.796,402.794,179.172,21.794,152.946
C03217=1097.525,408.043,402.755,179.175,21.801,152.947
C03218=1097.531,408.289,402.716,179.177,21.809,152.949
C03219=1097.537,408.536,402.676,179.180,21.817,152.950
C03220=1097.543,408.784,402.637,179.182,21.825,152.952
C03221=1097.548,409.030,402.598,179.185,21.832,152.953
C03222=1097.554,409.277,402.558,179.187,21.840,152.955
C03223=1097.561,409.524,402.518,179.190,21.848,152.956
C03224=1097.566,409.770,402.479,179.192,21.856,152.958
C03225=1097.572,410.017,402.439,179.195,21.864,152.960
C03226=1097.577,410.235,402.404,179.197,21.871,152.961
C03227=1097.582,410.453,402.369,179.199,21.878,152.962
C03228=1097.587,410.671,402.334,179.202,21.885,152.964
C03229=1097.593,410.888,402.299,179.204,21.892,152.965
C03230=1097.598,411.106,402.264,179.206,21.899,152.967
C03231=1097.603,411.324,402.229,179.208,21.906,152.968
C03232=1097.608,411.542,402.194,179.210,21.913,152.969
C03233=1097.614,411.760,402.159,179.213,21.921,152.971
C03234=1097.620,412.007,402.120,179.215,21.928,152.972
C03235=1097.625,412.253,402.080,179.218,21.937,152.974
C03236=1097.631,412.500,402.040,179.221,21.945,152.976
C03237=1097.637,412.747,402.001,179.223,21.954,152.977
C03238=1097.644,412.994,401.960,179.225,21.961,152.979
C03239=1097.649,413.240,401.921,179.228,21.969,152.981
C03240=1097.656,413.487,401.881,179.231,21.978,152.982
C03241=1097.661,413.733,401.841,179.233,21.986,152.984
C03242=1097.667,413.981,401.801,179.236,21.995,152.985
C03243=1097.674,414.227,401.761,179.239,22.003,152.987
C03244=1097.680,414.474,401.722,179.241,22.011,152.989
C03245=1097.686,414.720,401.682,179.243,22.020,152.991
C03246=1097.691,414.967,401.641,179.246,22.028,152.992
C03247=1097.697,415.214,401.602,179.249,22.036,152.994
C03248=1097.704,415.461,401.561,179.251,22.045,152.996
C03249=1097.710,415.707,401.521,179.254,22.054,152.997
C03250=1097.715,415.954,401.481,179.257,22.062,152.999
C03251=1097.722,416.201,401.441,179.259,22.070,153.001
C03252=1097.728,416.447,401.401,179.262,22.079,153.002
C03253=1097.734,416.694,401.360,179.264,22.087,153.004
C03254=1097.740,416.940,401.320,179.266,22.096,153.006
C03255=1097.745,417.188,401.280,179.269,22.105,153.008
C03256=1097.751,417.434,401.240,179.271,22.113,153.010
C03257=1097.757,417.681,401.200,179.274,22.123,153.011
C03258=1097.763,417.927,401.159,179.276,22.131,153.013
C03259=1097.770,418.174,401.119,179.279,22.140,153.015
C03260=1097.775,418.421,401.078,179.281,22.149,153.017
C03261=1097.782,418.667,401.038,179.284,22.158,153.019
C03262=1097.787,418.914,400.998,179.286,22.167,153.021
C03263=1097.794,419.161,400.957,179.289,22.175,153.022
C03264=1097.799,419.407,400.917,179.291,22.185,153.024
C03265=1097.804,419.654,400.876,179.294,22.194,153.026
C03266=1097.811,419.900,400.836,179.296,22.203,153.028
C03267=1097.816,420.147,400.795,179.299,22.212,153.030
C03268=1097.823,420.393,400.755,179.301,22.221,153.032
C03269=1097.828,420.640,400.715,179.304,22.230,153.034
C03270=1097.835,420.886,400.674,179.307,22.239,153.035
C03271=1097.841,421.133,400.633,179.309,22.249,153.037
C03272=1097.847,421.379,400.593,179.312,22.258,153.039
C03273=1097.853,421.626,400.552,179.314,22.267,153.041
C03274=1097.858,421.873,400.511,179.317,22.276,153.043
C03275=1097.866,422.120,400.470,179.319,22.285,153.045
C03276=1097.871,422.367,400.429,179.321,22.295,153.047
C03277=1097.878,422.613,400.389,179.324,22.304,153.049
C03278=1097.884,422.859,400.348,179.326,22.313,153.051
C03279=1097.889,423.106,400.307,179.329,22.323,153.053
C03280=1097.895,423.353,400.266,179.332,22.332,153.055
C03281=1097.902,423.599,400.225,179.334,22.342,153.057
C03282=1097.906,423.824,400.188,179.337,22.351,153.059
C03283=1097.912,424.048,400.150,179.338,22.359,153.061
C03284=1097.918,424.273,400.113,179.341,22.368,153.062
C03285=1097.923,424.498,400.076,179.342,22.377,153.064
C03286=1097.929,424.723,400.038,179.345,22.386,153.066
C03287=1097.934,424.948,400.001,179.347,22.395,153.068
C03288=1097.939,425.173,399.964,179.349,22.403,153.070
C03289=1097.945,425.397,399.926,179.352,22.412,153.072
C03290=1097.951,425.644,399.885,179.354,22.422,153.074
C03291=1097.957,425.890,399.844,179.357,22.432,153.076
C03292=1097.963,426.137,399.802,179.359,22.442,153.078
C03293=1097.969,426.383,399.762,179.361,22.452,153.080
C03294=1097.975,426.629,399.721,179.364,22.461,153.082
C03295=1097.981,426.876,399.679,179.367,22.471,153.084
C03296=1097.987,427.123,399.637,179.369,22.481,153.086
C03297=1097.993,427.369,399.597,179.371,22.491,153.089
C03298=1097.999,427.616,399.555,179.374,22.501,153.091
C03299=1098.005,427.862,399.514,179.376,22.511,153.093
C03300=1098.012,428.109,399.472,179.378,22.521,153.095
C03301=1098.017,428.355,399.430,179.380,22.531,153.097
C03302=1098.024,428.601,399.390,179.383,22.542,153.099
C03303=1098.030,428.848,399.349,179.385,22.552,153.102
C03304=1098.036,429.094,399.307,179.388,22.562,153.104
C03305=1098.042,429.341,399.265,179.390,22.572,153.106
C03306=1098.048,429.587,399.224,179.392,22.583,153.108
C03307=1098.053,429.833,399.182,179.395,22.593,153.111
C03308=1098.059,430.080,399.141,179.398,22.603,153.113
C03309=1098.066,430.327,399.099,179.400,22.614,153.115
C03310=1098.072,430.573,399.057,179.402,22.625,153.117
C03311=1098.078,430.819,399.016,179.404,22.635,153.120
C03312=1098.084,431.065,398.974,179.407,22.646,153.122
C03313=1098.091,431.311,398.932,179.409,22.656,153.124
C03314=1098.097,431.558,398.890,179.411,22.667,153.127
C03315=1098.103,431.804,398.849,179.414,22.677,153.129
C03316=1098.108,432.051,398.806,179.416,22.688,153.131
C03317=1098.114,432.297,398.765,179.419,22.699,153.134
C03318=1098.121,432.543,398.723,179.421,22.709,153.136
C03319=1098.127,432.790,398.681,179.423,22.721,153.138
C03320=1098.133,433.036,398.640,179.425,22.731,153.141
C03321=1098.139,433.282,398.598,179.428,22.742,153.143
C03322=1098.145,433.529,398.555,179.430,22.753,153.146
C03323=1098.151,433.775,398.513,179.433,22.764,153.148
C03324=1098.157,434.020,398.471,179.435,22.775,153.150
C03325=1098.163,434.267,398.429,179.437,22.786,153.153
C03326=1098.169,434.514,398.387,179.439,22.797,153.155
C03327=1098.175,434.759,398.345,179.442,22.809,153.158
C03328=1098.181,435.006,398.303,179.444,22.819,153.160
C03329=1098.187,435.252,398.261,179.446,22.831,153.163
C03330=1098.193,435.499,398.219,179.449,22.842,153.165
C03331=1098.199,435.745,398.176,179.451,22.853,153.168
C03332=1098.206,435.991,398.134,179.453,22.865,153.170
C03333=1098.211,436.237,398.092,179.455,22.876,153.173
C03334=1098.218,436.483,398.049,179.458,22.888,153.175
C03335=1098.223,436.729,398.007,179.460,22.899,153.178
C03336=1098.230,436.976,397.965,179.462,22.910,153.180
C03337=1098.235,437.222,397.922,179.465,22.922,153.183
C03338=1098.244,437.531,397.869,179.467,22.936,153.186
C03339=1098.251,437.840,397.816,179.471,22.952,153.190
C03340=1098.259,438.149,397.762,179.473,22.966,153.193
C03341=1098.266,438.457,397.709,179.475,22.981,153.196
C03342=1098.273,438.704,397.667,179.478,22.993,153.199
C03343=1098.278,438.950,397.624,179.480,23.005,153.202
C03344=1098.285,439.197,397.582,179.482,23.016,153.204
C03345=1098.291,439.442,397.539,179.485,23.028,153.207
C03346=1098.298,439.689,397.496,179.487,23.040,153.209
C03347=1098.303,439.935,397.453,179.490,23.052,153.212
C03348=1098.310,440.181,397.411,179.491,23.064,153.215
C03349=1098.316,440.427,397.368,179.494,23.076,153.218
C03350=1098.322,440.673,397.326,179.496,23.088,153.220
C03351=1098.329,440.920,397.282,179.498,23.101,153.223
C03352=1098.334,441.166,397.240,179.500,23.112,153.226
C03353=1098.340,441.412,397.197,179.502,23.125,153.229
C03354=1098.347,441.657,397.154,179.505,23.138,153.232
C03355=1098.353,441.904,397.111,179.507,23.150,153.234
C03356=1098.359,442.150,397.067,179.509,23.162,153.237
C03357=1098.365,442.396,397.025,179.511,23.175,153.240
C03358=1098.372,442.642,396.981,179.513,23.187,153.243
C03359=1098.377,442.888,396.939,179.515,23.200,153.246
C03360=1098.383,443.134,396.895,179.518,23.212,153.249
C03361=1098.389,443.381,396.852,179.520,23.225,153.252
C03362=1098.396,443.626,396.809,179.522,23.238,153.255
C03363=1098.402,443.872,396.766,179.524,23.250,153.257
C03364=1098.409,444.118,396.722,179.526,23.263,153.261
C03365=1098.414,444.364,396.680,179.528,23.276,153.263
C03366=1098.420,444.610,396.636,179.529,23.289,153.266
C03367=1098.427,444.857,396.593,179.530,23.302,153.270
C03368=1098.433,445.102,396.550,179.532,23.314,153.272
C03369=1098.439,445.348,396.507,179.533,23.327,153.275
C03370=1098.446,445.594,396.463,179.533,23.339,153.279
C03371=1098.452,445.841,396.420,179.535,23.352,153.282
C03372=1098.458,446.086,396.376,179.535,23.364,153.285
C03373=1098.464,446.333,396.333,179.535,23.377,153.288
C03374=1098.470,446.579,396.289,179.536,23.390,153.291
C03375=1098.477,446.825,396.245,179.537,23.403,153.294
C03376=1098.482,447.071,396.203,179.536,23.415,153.297
C03377=1098.489,447.317,396.159,179.536,23.428,153.301
C03378=1098.495,447.563,396.116,179.536,23.440,153.304
C03379=1098.501,447.809,396.072,179.536,23.452,153.307
C03380=1098.507,448.055,396.028,179.535,23.465,153.310
C03381=1098.513,448.301,395.984,179.535,23.478,153.314
C03382=1098.519,448.547,395.941,179.534,23.490,153.317
C03383=1098.525,448.793,395.897,179.534,23.503,153.320
C03384=1098.532,449.039,395.853,179.532,23.515,153.323
C03385=1098.538,449.285,395.809,179.531,23.527,153.327
C03386=1098.544,449.532,395.766,179.531,23.540,153.330
C03387=1098.550,449.777,395.723,179.529,23.552,153.333
C03388=1098.556,450.023,395.679,179.528,23.565,153.337
C03389=1098.563,450.269,395.635,179.527,23.577,153.340
C03390=1098.168,450.262,395.480,179.465,23.794,153.403
C03391=1098.161,450.016,395.524,179.467,23.782,153.400
C03392=1098.155,449.769,395.567,179.468,23.769,153.397
C03393=1098.149,449.523,395.611,179.469,23.757,153.393
C03394=1098.143,449.277,395.655,179.470,23.744,153.390
C03395=1098.137,449.031,395.699,179.471,23.732,153.387
C03396=1098.130,448.785,395.743,179.472,23.719,153.384
C03397=1098.124,448.540,395.786,179.473,23.707,153.380
C03398=1098.118,448.294,395.830,179.473,23.694,153.377
C03399=1098.112,448.047,395.873,179.474,23.682,153.374
C03400=1098.105,447.801,395.917,179.473,23.669,153.370
C03401=1098.099,447.555,395.961,179.474,23.656,153.367
C03402=1098.093,447.309,396.005,179.474,23.644,153.364
C03403=1098.087,447.064,396.048,179.474,23.631,153.361
C03404=1098.081,446.817,396.091,179.474,23.619,153.358
C03405=1098.074,446.571,396.135,179.474,23.606,153.355
C03406=1098.068,446.326,396.179,179.473,23.593,153.351
C03407=1098.062,446.079,396.222,179.473,23.581,153.348
C03408=1098.056,445.834,396.266,179.472,23.568,153.345
C03409=1098.049,445.588,396.310,179.471,23.555,153.342
C03410=1098.043,445.341,396.353,179.470,23.542,153.339
C03411=1098.037,445.095,396.397,179.469,23.529,153.336
C03412=1098.031,444.849,396.440,179.467,23.517,153.333
C03413=1098.025,444.603,396.483,179.466,23.504,153.330
C03414=1098.019,444.357,396.526,179.465,23.491,153.327
C03415=1098.012,444.111,396.570,179.462,23.479,153.324
C03416=1098.007,443.865,396.613,179.461,23.466,153.321
C03417=1098.000,443.619,396.656,179.458,23.453,153.318
C03418=1097.994,443.373,396.699,179.456,23.440,153.315
C03419=1097.988,443.127,396.743,179.454,23.427,153.312
C03420=1097.982,442.881,396.786,179.452,23.414,153.309
C03421=1097.976,442.634,396.829,179.450,23.402,153.306
C03422=1097.970,442.389,396.873,179.448,23.389,153.303
C03423=1097.963,442.143,396.915,179.445,23.377,153.300
C03424=1097.957,441.896,396.958,179.443,23.364,153.298
C03425=1097.951,441.651,397.002,179.440,23.352,153.295
C03426=1097.944,441.404,397.044,179.438,23.339,153.292
C03427=1097.939,441.158,397.087,179.436,23.327,153.289
C03428=1097.932,440.912,397.130,179.434,23.315,153.286
C03429=1097.926,440.665,397.173,179.431,23.302,153.284
C03430=1097.920,440.420,397.215,179.429,23.290,153.281
C03431=1097.914,440.174,397.259,179.427,23.278,153.278
C03432=1097.907,439.928,397.301,179.425,23.266,153.275
C03433=1097.901,439.682,397.345,179.422,23.254,153.273
C03434=1097.894,439.435,397.387,179.420,23.242,153.270
C03435=1097.889,439.189,397.430,179.418,23.230,153.267
C03436=1097.883,438.943,397.473,179.416,23.218,153.264
C03437=1097.877,438.697,397.515,179.413,23.206,153.262
C03438=1097.870,438.451,397.558,179.411,23.194,153.259
C03439=1097.863,438.151,397.610,179.408,23.180,153.256
C03440=1097.855,437.849,397.661,179.405,23.165,153.253
C03441=1097.848,437.549,397.713,179.402,23.151,153.250
C03442=1097.840,437.249,397.765,179.400,23.137,153.246
C03443=1097.834,437.002,397.808,179.398,23.125,153.244
C03444=1097.828,436.757,397.850,179.395,23.114,153.241
C03445=1097.822,436.510,397.893,179.393,23.102,153.239
C03446=1097.816,436.264,397.935,179.391,23.091,153.236
C03447=1097.809,436.018,397.977,179.388,23.079,153.234
C03448=1097.803,435.772,398.020,179.385,23.068,153.231
C03449=1097.798,435.526,398.062,179.383,23.057,153.228
C03450=1097.791,435.279,398.105,179.381,23.045,153.226
C03451=1097.785,435.033,398.146,179.379,23.034,153.223
C03452=1097.779,434.787,398.189,179.376,23.023,153.221
C03453=1097.773,434.541,398.231,179.374,23.011,153.218
C03454=1097.767,434.294,398.273,179.372,23.000,153.216
C03455=1097.761,434.048,398.316,179.370,22.989,153.214
C03456=1097.755,433.802,398.357,179.367,22.978,153.211
C03457=1097.749,433.555,398.399,179.365,22.967,153.209
C03458=1097.743,433.309,398.442,179.362,22.955,153.206
C03459=1097.737,433.063,398.484,179.360,22.945,153.204
C03460=1097.731,432.817,398.526,179.357,22.934,153.201
C03461=1097.724,432.570,398.568,179.355,22.923,153.199
C03462=1097.718,432.324,398.609,179.353,22.912,153.197
C03463=1097.713,432.077,398.651,179.350,22.902,153.194
C03464=1097.706,431.831,398.694,179.348,22.891,153.192
C03465=1097.700,431.585,398.735,179.346,22.880,153.190
C03466=1097.694,431.339,398.776,179.343,22.869,153.187
C03467=1097.688,431.092,398.818,179.341,22.859,153.185
C03468=1097.682,430.846,398.860,179.338,22.848,153.183
C03469=1097.676,430.600,398.902,179.336,22.837,153.180
C03470=1097.670,430.353,398.944,179.334,22.827,153.178
C03471=1097.664,430.107,398.986,179.331,22.816,153.176
C03472=1097.658,429.860,399.027,179.328,22.806,153.173
C03473=1097.652,429.614,399.069,179.326,22.796,153.171
C03474=1097.645,429.367,399.111,179.323,22.785,153.169
C03475=1097.639,429.121,399.152,179.321,22.775,153.167
C03476=1097.633,428.875,399.193,179.318,22.764,153.164
C03477=1097.628,428.629,399.235,179.316,22.754,153.162
C03478=1097.621,428.382,399.277,179.314,22.744,153.160
C03479=1097.615,428.136,399.318,179.311,22.733,153.158
C03480=1097.609,427.889,399.360,179.309,22.723,153.156
C03481=1097.603,427.643,399.401,179.306,22.713,153.154
C03482=1097.597,427.396,399.442,179.304,22.703,153.151
C03483=1097.591,427.149,399.484,179.301,22.693,153.149
C03484=1097.584,426.904,399.525,179.299,22.683,153.147
C03485=1097.578,426.657,399.566,179.297,22.673,153.145
C03486=1097.572,426.411,399.607,179.294,22.663,153.143
C03487=1097.566,426.164,399.649,179.291,22.653,153.141
C03488=1097.560,425.917,399.690,179.289,22.643,153.139
C03489=1097.554,425.671,399.731,179.287,22.633,153.136
C03490=1097.549,425.424,399.772,179.284,22.623,153.134
C03491=1097.543,425.200,399.810,179.282,22.615,153.132
C03492=1097.537,424.974,399.847,179.280,22.606,153.131
C03493=1097.532,424.749,399.885,179.277,22.597,153.129
C03494=1097.526,424.524,399.922,179.275,22.588,153.127
C03495=1097.521,424.299,399.961,179.273,22.579,153.125
C03496=1097.515,424.074,399.998,179.270,22.570,153.123
C03497=1097.510,423.849,400.035,179.268,22.562,153.121
C03498=1097.504,423.623,400.073,179.266,22.553,153.119
C03499=1097.498,423.377,400.114,179.263,22.543,153.117
C03500=1097.492,423.130,400.154,179.261,22.534,153.115
C03501=1097.486,422.884,400.196,179.259,22.524,153.113
C03502=1097.481,422.637,400.237,179.256,22.515,153.111
C03503=1097.474,422.390,400.277,179.253,22.505,153.109
C03504=1097.468,422.144,400.318,179.251,22.496,153.107
C03505=1097.462,421.898,400.358,179.248,22.486,153.105
C03506=1097.456,421.651,400.399,179.246,22.477,153.104
C03507=1097.450,421.405,400.440,179.243,22.468,153.102
C03508=1097.444,421.158,400.481,179.241,22.459,153.100
C03509=1097.438,420.911,400.521,179.238,22.449,153.098
C03510=1097.432,420.665,400.562,179.236,22.440,153.096
C03511=1097.426,420.418,400.602,179.233,22.431,153.094
C03512=1097.420,420.172,400.644,179.231,22.422,153.092
C03513=1097.414,419.925,400.684,179.229,22.413,153.090
C03514=1097.408,419.678,400.725,179.226,22.404,153.088
C03515=1097.402,419.432,400.765,179.223,22.395,153.086
C03516=1097.396,419.185,400.805,179.221,22.386,153.085
C03517=1097.390,418.939,400.846,179.218,22.377,153.083
C03518=1097.384,418.692,400.886,179.216,22.368,153.081
C03519=1097.378,418.445,400.927,179.213,22.359,153.079
C03520=1097.372,418.198,400.967,179.211,22.350,153.077
C03521=1097.366,417.952,401.007,179.208,22.341,153.075
C03522=1097.360,417.705,401.048,179.205,22.332,153.074
C03523=1097.354,417.459,401.088,179.203,22.323,153.072
C03524=1097.348,417.212,401.129,179.200,22.314,153.070
C03525=1097.342,416.965,401.169,179.198,22.306,153.068
C03526=1097.337,416.719,401.210,179.195,22.297,153.067
C03527=1097.330,416.473,401.250,179.193,22.288,153.065
C03528=1097.324,416.226,401.289,179.190,22.279,153.063
C03529=1097.319,415.979,401.330,179.187,22.271,153.061
C03530=1097.312,415.732,401.370,179.185,22.262,153.059
C03531=1097.306,415.486,401.410,179.182,22.254,153.058
C03532=1097.299,415.239,401.450,179.179,22.245,153.056
C03533=1097.294,414.992,401.490,179.177,22.237,153.054
C03534=1097.288,414.745,401.531,179.175,22.228,153.053
C03535=1097.281,414.499,401.571,179.172,22.220,153.051
C03536=1097.275,414.252,401.610,179.169,22.211,153.049
C03537=1097.270,414.005,401.650,179.167,22.203,153.047
C03538=1097.264,413.758,401.690,179.164,22.195,153.046
C03539=1097.258,413.512,401.730,179.161,22.186,153.044
C03540=1097.251,413.265,401.770,179.159,22.178,153.043
C03541=1097.245,413.018,401.810,179.156,22.170,153.041
C03542=1097.240,412.771,401.850,179.154,22.161,153.039
C03543=1097.234,412.525,401.889,179.151,22.153,153.038
C03544=1097.228,412.278,401.930,179.148,22.145,153.036
C03545=1097.222,412.031,401.969,179.146,22.137,153.034
C03546=1097.215,411.785,402.009,179.143,22.129,153.033
C03547=1097.210,411.567,402.044,179.141,22.121,153.031
C03548=1097.206,411.348,402.079,179.139,22.114,153.030
C03549=1097.200,411.130,402.114,179.137,22.107,153.028
C03550=1097.195,410.912,402.150,179.135,22.100,153.027
C03551=1097.190,410.694,402.185,179.132,22.092,153.026
C03552=1097.185,410.476,402.220,179.129,22.086,153.024
C03553=1097.179,410.257,402.254,179.127,22.078,153.023
C03554=1097.174,410.039,402.289,179.125,22.071,153.021
C03555=1097.168,409.792,402.329,179.123,22.064,153.020
C03556=1097.163,409.546,402.369,179.120,22.055,153.018
C03557=1097.157,409.299,402.409,179.117,22.048,153.017
C03558=1097.150,409.052,402.448,179.115,22.040,153.015
C03559=1097.145,408.805,402.487,179.112,22.032,153.014
C03560=1097.139,408.559,402.527,179.109,22.024,153.012
C03561=1097.133,408.312,402.567,179.107,22.016,153.010
C03562=1097.127,408.065,402.606,179.104,22.008,153.009
C03563=1097.121,407.818,402.645,179.101,22.000,153.007
C03564=1097.115,407.571,402.685,179.099,21.993,153.006
C03565=1097.109,407.324,402.724,179.096,21.985,153.004
C03566=1097.103,407.077,402.763,179.093,21.977,153.003
C03567=1097.098,406.831,402.802,179.091,21.970,153.001
C03568=1097.092,406.584,402.842,179.089,21.962,153.000
C03569=1097.085,406.337,402.880,179.086,21.955,152.999
C03570=1097.080,406.091,402.919,179.083,21.947,152.997
C03571=1097.073,405.843,402.959,179.080,21.939,152.996
C03572=1097.067,405.596,402.998,179.078,21.932,152.994
C03573=1097.062,405.350,403.037,179.075,21.924,152.993
C03574=1097.056,405.103,403.077,179.073,21.917,152.991
C03575=1097.050,404.856,403.116,179.070,21.909,152.990
C03576=1097.044,404.609,403.155,179.068,21.902,152.988
C03577=1097.038,404.362,403.193,179.065,21.895,152.987
C03578=1097.032,404.115,403.233,179.063,21.887,152.986
C03579=1097.026,403.868,403.272,179.060,21.880,152.984
C03580=1097.020,403.622,403.310,179.057,21.873,152.983
C03581=1097.014,403.375,403.350,179.054,21.865,152.981
C03582=1097.009,403.128,403.388,179.052,21.858,152.980
C03583=1097.003,402.881,403.428,179.049,21.850,152.979
C03584=1096.997,402.635,403.466,179.047,21.844,152.977
C03585=1096.990,402.387,403.506,179.044,21.836,152.976
C03586=1096.985,402.140,403.544,179.042,21.829,152.975
C03587=1096.978,401.894,403.583,179.038,21.822,152.973
C03588=1096.973,401.646,403.621,179.036,21.815,152.972
C03589=1096.967,401.399,403.661,179.033,21.807,152.971
C03590=1096.961,401.153,403.699,179.031,21.800,152.969
C03591=1096.955,400.905,403.738,179.028,21.793,152.968
C03592=1096.949,400.659,403.776,179.025,21.786,152.967
C03593=1096.943,400.412,403.815,179.023,21.779,152.965
C03594=1096.938,400.165,403.854,179.020,21.772,152.964
C03595=1096.931,399.918,403.892,179.018,21.765,152.963
C03596=1096.926,399.671,403.931,179.014,21.758,152.961
C03597=1096.920,399.424,403.969,179.012,21.751,152.960
C03598=1096.914,399.177,404.008,179.010,21.744,152.959
C03599=1096.908,398.931,404.046,179.006,21.737,152.958
C03600=1096.902,398.683,404.086,179.004,21.730,152.956
C03601=1096.896,398.437,404.123,179.001,21.723,152.955
C03602=1096.891,398.190,404.162,178.999,21.716,152.954
C03603=1096.885,397.971,404.195,178.996,21.710,152.953
C03604=1096.880,397.754,404.230,178.994,21.705,152.952
C03605=1096.874,397.536,404.264,178.992,21.698,152.950
C03606=1096.869,397.318,404.297,178.989,21.692,152.949
C03607=1096.864,397.100,404.332,178.986,21.686,152.948
C03608=1096.859,396.882,404.366,178.985,21.681,152.947
C03609=1096.854,396.664,404.399,178.982,21.674,152.946
C03610=1096.849,396.446,404.433,178.979,21.668,152.945
C03611=1096.843,396.199,404.471,178.977,21.662,152.944
C03612=1096.838,395.952,404.509,178.975,21.655,152.943
C03613=1096.831,395.705,404.547,178.971,21.648,152.941
C03614=1096.825,395.458,404.586,178.969,21.642,152.940
C03615=1096.820,395.211,404.624,178.966,21.636,152.939
C03616=1096.813,394.964,404.662,178.964,21.629,152.938
C03617=1096.807,394.717,404.700,178.961,21.622,152.937
C03618=1096.802,394.470,404.738,178.958,21.616,152.935
C03619=1096.796,394.223,404.777,178.956,21.609,152.934
C03620=1096.790,393.976,404.814,178.952,21.603,152.933
C03621=1096.784,393.729,404.852,178.950,21.596,152.932
C03622=1096.779,393.482,404.890,178.947,21.590,152.931
C03623=1096.772,393.235,404.929,178.945,21.584,152.930
C03624=1096.766,392.988,404.966,178.942,21.577,152.929
C03625=1096.760,392.741,405.004,178.939,21.570,152.927
C03626=1096.755,392.494,405.042,178.936,21.564,152.926
C03627=1096.749,392.247,405.080,178.934,21.558,152.925
C03628=1096.743,392.000,405.118,178.931,21.552,152.924
C03629=1096.737,391.753,405.156,178.928,21.545,152.923
C03630=1096.731,391.507,405.194,178.925,21.539,152.922
C03631=1096.725,391.260,405.232,178.923,21.532,152.921
C03632=1096.719,391.012,405.270,178.920,21.526,152.920
C03633=1096.713,390.766,405.307,178.917,21.520,152.919
C03634=1096.707,390.518,405.344,178.914,21.514,152.918
C03635=1096.701,390.271,405.382,178.912,21.508,152.916
C03636=1096.695,390.025,405.420,178.909,21.501,152.915
C03637=1096.689,389.778,405.458,178.906,21.495,152.914
C03638=1096.683,389.531,405.496,178.903,21.489,152.913
C03639=1096.677,389.283,405.533,178.900,21.483,152.912
C03640=1096.671,389.036,405.571,178.898,21.477,152.911
